LIN {X 0,Y 476.575,Z 542.325,A -85,B 0,C 180,E1 -7304.355,E2 -7304.355} C_VEL
LIN {X 0,Y 476.998,Z 529.723,A -85,B 0,C 180,E1 -7304.805,E2 -7304.805} C_VEL
LIN {X 0,Y 477.328,Z 516.997,A -85,B 0,C 180,E1 -7305.095,E2 -7305.095} C_VEL
LIN {X 0,Y 477.658,Z 432.911,A -85,B 0,C 180,E1 -7306.37,E2 -7306.37} C_VEL
LIN {X 0,Y 475.32,Z 411.409,A -85,B 0,C 180,E1 -7306.785,E2 -7306.785} C_VEL
LIN {X 0,Y 475.32,Z 409.484,A -85,B 0,C 180,E1 -7306.979,E2 -7306.979} C_VEL
LIN {X 0,Y 476.001,Z 385.629,A -85,B 0,C 180,E1 -7310.076,E2 -7310.076} C_VEL
LIN {X 0,Y 476.795,Z 363.158,A -85,B 0,C 180,E1 -7312.992,E2 -7312.992} C_VEL
LIN {X 0,Y 477.623,Z 341.029,A -85,B 0,C 180,E1 -7315.89,E2 -7315.89} C_VEL
LIN {X 0,Y 478.026,Z 328.359,A -85,B 0,C 180,E1 -7317.578,E2 -7317.578} C_VEL
LIN {X 0,Y 474.979,Z 313.924,A -85,B 0,C 180,E1 -7319.714,E2 -7319.714} C_VEL
LIN {X 0,Y 474.64,Z 312.462,A -85,B 0,C 180,E1 -7319.982,E2 -7319.982} C_VEL
LIN {X 0,Y 474.612,Z 312.36,A -85,B 0,C 180,E1 -7323.222,E2 -7323.222} C_VEL
LIN {X 0,Y 474.569,Z 312.369,A -85,B 0,C 180,E1 -7326.325,E2 -7326.325} C_VEL
LIN {X 0,Y 474.597,Z 312.358,A -85,B 0,C 180,E1 -7329.643,E2 -7329.643} C_VEL
LIN {X 0,Y 474.565,Z 312.367,A -85,B 0,C 180,E1 -7332.939,E2 -7332.939} C_VEL
LIN {X 0,Y 474.598,Z 312.354,A -85,B 0,C 180,E1 -7335.894,E2 -7335.894} C_VEL
LIN {X 0,Y 474.596,Z 312.364,A -85,B 0,C 180,E1 -7339.044,E2 -7339.044} C_VEL
LIN {X 0,Y 474.584,Z 312.349,A -85,B 0,C 180,E1 -7341.707,E2 -7341.707} C_VEL
LIN {X 0,Y 474.606,Z 312.35,A -85,B 0,C 180,E1 -7344.724,E2 -7344.724} C_VEL
LIN {X 0,Y 474.621,Z 312.366,A -85,B 0,C 180,E1 -7347.787,E2 -7347.787} C_VEL
LIN {X 0,Y 474.6,Z 312.355,A -85,B 0,C 180,E1 -7350.888,E2 -7350.888} C_VEL
LIN {X 0,Y 474.584,Z 312.366,A -85,B 0,C 180,E1 -7353.624,E2 -7353.624} C_VEL
LIN {X 0,Y 474.627,Z 312.357,A -85,B 0,C 180,E1 -7356.642,E2 -7356.642} C_VEL
LIN {X 0,Y 474.645,Z 312.353,A -85,B 0,C 180,E1 -7360.089,E2 -7360.089} C_VEL
LIN {X 0,Y 474.626,Z 312.359,A -85,B 0,C 180,E1 -7362.774,E2 -7362.774} C_VEL
LIN {X 0,Y 474.637,Z 312.361,A -85,B 0,C 180,E1 -7365.421,E2 -7365.421} C_VEL
LIN {X 0,Y 474.696,Z 312.353,A -85,B 0,C 180,E1 -7368.037,E2 -7368.037} C_VEL
LIN {X 0,Y 474.693,Z 312.356,A -85,B 0,C 180,E1 -7371.486,E2 -7371.486} C_VEL
LIN {X 0,Y 474.749,Z 312.343,A -85,B 0,C 180,E1 -7374.052,E2 -7374.052} C_VEL
LIN {X 0,Y 474.863,Z 312.335,A -85,B 0,C 180,E1 -7377.455,E2 -7377.455} C_VEL
LIN {X 0,Y 474.869,Z 312.325,A -85,B 0,C 180,E1 -7380,E2 -7380} C_VEL
LIN {X 0,Y 474.872,Z 312.326,A -85,B 0,C 180,E1 -7382.545,E2 -7382.545} C_VEL
LIN {X 0,Y 474.73,Z 312.346,A -85,B 0,C 180,E1 -7385.948,E2 -7385.948} C_VEL
LIN {X 0,Y 474.699,Z 312.345,A -85,B 0,C 180,E1 -7388.514,E2 -7388.514} C_VEL
LIN {X 0,Y 474.696,Z 312.352,A -85,B 0,C 180,E1 -7391.963,E2 -7391.963} C_VEL
LIN {X 0,Y 474.671,Z 312.357,A -85,B 0,C 180,E1 -7395.767,E2 -7395.767} C_VEL
LIN {X 0,Y 474.652,Z 312.357,A -85,B 0,C 180,E1 -7399.011,E2 -7399.011} C_VEL
LIN {X 0,Y 474.58,Z 312.368,A -85,B 0,C 180,E1 -7401.729,E2 -7401.729} C_VEL
LIN {X 0,Y 474.619,Z 312.36,A -85,B 0,C 180,E1 -7404.495,E2 -7404.495} C_VEL
LIN {X 0,Y 474.592,Z 312.36,A -85,B 0,C 180,E1 -7407.327,E2 -7407.327} C_VEL
LIN {X 0,Y 474.582,Z 312.348,A -85,B 0,C 180,E1 -7410.232,E2 -7410.232} C_VEL
LIN {X 0,Y 474.609,Z 312.362,A -85,B 0,C 180,E1 -7413.223,E2 -7413.223} C_VEL
LIN {X 0,Y 474.577,Z 312.363,A -85,B 0,C 180,E1 -7416.325,E2 -7416.325} C_VEL
LIN {X 0,Y 474.596,Z 312.354,A -85,B 0,C 180,E1 -7419.644,E2 -7419.644} C_VEL
LIN {X 0,Y 474.564,Z 312.369,A -85,B 0,C 180,E1 -7422.94,E2 -7422.94} C_VEL
LIN {X 0,Y 474.576,Z 312.358,A -85,B 0,C 180,E1 -7425.892,E2 -7425.892} C_VEL
LIN {X 0,Y 474.596,Z 312.364,A -85,B 0,C 180,E1 -7429.046,E2 -7429.046} C_VEL
LIN {X 0,Y 474.594,Z 312.36,A -85,B 0,C 180,E1 -7431.707,E2 -7431.707} C_VEL
LIN {X 0,Y 474.616,Z 312.362,A -85,B 0,C 180,E1 -7434.726,E2 -7434.726} C_VEL
LIN {X 0,Y 474.615,Z 312.362,A -85,B 0,C 180,E1 -7437.787,E2 -7437.787} C_VEL
LIN {X 0,Y 474.592,Z 312.366,A -85,B 0,C 180,E1 -7440.892,E2 -7440.892} C_VEL
LIN {X 0,Y 474.571,Z 312.359,A -85,B 0,C 180,E1 -7443.624,E2 -7443.624} C_VEL
LIN {X 0,Y 474.634,Z 312.361,A -85,B 0,C 180,E1 -7446.643,E2 -7446.643} C_VEL
LIN {X 0,Y 474.647,Z 312.359,A -85,B 0,C 180,E1 -7450.09,E2 -7450.09} C_VEL
LIN {X 0,Y 474.625,Z 312.333,A -85,B 0,C 180,E1 -7451.631,E2 -7451.631} C_VEL
LIN {X 0,Y 474.463,Z 312.988,A -85,B 0,C 180,E1 -7452.075,E2 -7452.075} C_VEL
LIN {X 0,Y 474.092,Z 314.652,A -85,B 0,C 180,E1 -7452.481,E2 -7452.481} C_VEL
LIN {X 0,Y 473.329,Z 318.415,A -85,B 0,C 180,E1 -7453.005,E2 -7453.005} C_VEL
LIN {X 0,Y 472.491,Z 323.287,A -85,B 0,C 180,E1 -7453.422,E2 -7453.422} C_VEL
LIN {X 0,Y 471.778,Z 328.831,A -85,B 0,C 180,E1 -7453.729,E2 -7453.729} C_VEL
LIN {X 0,Y 471.44,Z 334.777,A -85,B 0,C 180,E1 -7453.9,E2 -7453.9} C_VEL
LIN {X 0,Y 471.117,Z 394.353,A -85,B 0,C 180,E1 -7454.84,E2 -7454.84} C_VEL
LIN {X 0,Y 470.981,Z 407.411,A -85,B 0,C 180,E1 -7455.222,E2 -7455.222} C_VEL
LIN {X 0,Y 470.798,Z 419.402,A -85,B 0,C 180,E1 -7455.741,E2 -7455.741} C_VEL
LIN {X 0,Y 470.507,Z 431.055,A -85,B 0,C 180,E1 -7456.419,E2 -7456.419} C_VEL
LIN {X 0,Y 470.005,Z 442.247,A -85,B 0,C 180,E1 -7457.258,E2 -7457.258} C_VEL
LIN {X 0,Y 469.55,Z 452.592,A -85,B 0,C 180,E1 -7458.233,E2 -7458.233} C_VEL
LIN {X 0,Y 469.181,Z 461.025,A -85,B 0,C 180,E1 -7459.208,E2 -7459.208} C_VEL
LIN {X 0,Y 468.744,Z 468.789,A -85,B 0,C 180,E1 -7460.289,E2 -7460.289} C_VEL
LIN {X 0,Y 468.373,Z 476.47,A -85,B 0,C 180,E1 -7461.609,E2 -7461.609} C_VEL
LIN {X 0,Y 468.091,Z 482.229,A -85,B 0,C 180,E1 -7462.84,E2 -7462.84} C_VEL
LIN {X 0,Y 467.937,Z 486.507,A -85,B 0,C 180,E1 -7463.965,E2 -7463.965} C_VEL
LIN {X 0,Y 467.639,Z 490.4,A -85,B 0,C 180,E1 -7465.259,E2 -7465.259} C_VEL
LIN {X 0,Y 467.443,Z 493.271,A -85,B 0,C 180,E1 -7466.552,E2 -7466.552} C_VEL
LIN {X 0,Y 467.481,Z 494.631,A -85,B 0,C 180,E1 -7467.415,E2 -7467.415} C_VEL
LIN {X 0,Y 467.356,Z 495.617,A -85,B 0,C 180,E1 -7468.277,E2 -7468.277} C_VEL
LIN {X 0,Y 467.433,Z 496.204,A -85,B 0,C 180,E1 -7469.139,E2 -7469.139} C_VEL
LIN {X 0,Y 467.417,Z 496.436,A -85,B 0,C 180,E1 -7470,E2 -7470} C_VEL
LIN {X 0,Y 467.433,Z 496.253,A -85,B 0,C 180,E1 -7470.861,E2 -7470.861} C_VEL
LIN {X 0,Y 467.356,Z 495.698,A -85,B 0,C 180,E1 -7471.723,E2 -7471.723} C_VEL
LIN {X 0,Y 467.48,Z 494.743,A -85,B 0,C 180,E1 -7472.585,E2 -7472.585} C_VEL
LIN {X 0,Y 467.437,Z 493.435,A -85,B 0,C 180,E1 -7473.448,E2 -7473.448} C_VEL
LIN {X 0,Y 467.634,Z 490.625,A -85,B 0,C 180,E1 -7474.741,E2 -7474.741} C_VEL
LIN {X 0,Y 467.927,Z 486.808,A -85,B 0,C 180,E1 -7476.035,E2 -7476.035} C_VEL
LIN {X 0,Y 468.063,Z 481.73,A -85,B 0,C 180,E1 -7477.377,E2 -7477.377} C_VEL
LIN {X 0,Y 468.507,Z 474.508,A -85,B 0,C 180,E1 -7478.845,E2 -7478.845} C_VEL
LIN {X 0,Y 468.968,Z 466.485,A -85,B 0,C 180,E1 -7480.142,E2 -7480.142} C_VEL
LIN {X 0,Y 469.344,Z 458.267,A -85,B 0,C 180,E1 -7481.225,E2 -7481.225} C_VEL
LIN {X 0,Y 469.747,Z 449.245,A -85,B 0,C 180,E1 -7482.2,E2 -7482.2} C_VEL
LIN {X 0,Y 470.256,Z 438.755,A -85,B 0,C 180,E1 -7483.114,E2 -7483.114} C_VEL
LIN {X 0,Y 470.569,Z 427.264,A -85,B 0,C 180,E1 -7483.914,E2 -7483.914} C_VEL
LIN {X 0,Y 470.826,Z 416.033,A -85,B 0,C 180,E1 -7484.517,E2 -7484.517} C_VEL
LIN {X 0,Y 471.032,Z 402.87,A -85,B 0,C 180,E1 -7485.025,E2 -7485.025} C_VEL
LIN {X 0,Y 471.056,Z 389.173,A -85,B 0,C 180,E1 -7485.356,E2 -7485.356} C_VEL
LIN {X 0,Y 471.439,Z 324.141,A -85,B 0,C 180,E1 -7486.359,E2 -7486.359} C_VEL
LIN {X 0,Y 467.78,Z 314.282,A -85,B 0,C 180,E1 -7486.672,E2 -7486.672} C_VEL
LIN {X 0,Y 467.575,Z 313.366,A -85,B 0,C 180,E1 -7486.826,E2 -7486.826} C_VEL
LIN {X 0,Y 467.589,Z 313.223,A -85,B 0,C 180,E1 -7489.309,E2 -7489.309} C_VEL
LIN {X 0,Y 467.529,Z 313.235,A -85,B 0,C 180,E1 -7492.074,E2 -7492.074} C_VEL
LIN {X 0,Y 467.549,Z 313.246,A -85,B 0,C 180,E1 -7494.89,E2 -7494.89} C_VEL
LIN {X 0,Y 467.54,Z 313.225,A -85,B 0,C 180,E1 -7497.774,E2 -7497.774} C_VEL
LIN {X 0,Y 467.534,Z 313.246,A -85,B 0,C 180,E1 -7501.037,E2 -7501.037} C_VEL
LIN {X 0,Y 467.563,Z 313.241,A -85,B 0,C 180,E1 -7504.237,E2 -7504.237} C_VEL
LIN {X 0,Y 467.519,Z 313.239,A -85,B 0,C 180,E1 -7507.181,E2 -7507.181} C_VEL
LIN {X 0,Y 467.553,Z 313.244,A -85,B 0,C 180,E1 -7510.266,E2 -7510.266} C_VEL
LIN {X 0,Y 467.513,Z 313.241,A -85,B 0,C 180,E1 -7512.568,E2 -7512.568} C_VEL
LIN {X 0,Y 467.558,Z 313.243,A -85,B 0,C 180,E1 -7515.051,E2 -7515.051} C_VEL
LIN {X 0,Y 467.555,Z 313.239,A -85,B 0,C 180,E1 -7518.725,E2 -7518.725} C_VEL
LIN {X 0,Y 467.546,Z 313.229,A -85,B 0,C 180,E1 -7521.953,E2 -7521.953} C_VEL
LIN {X 0,Y 467.548,Z 313.243,A -85,B 0,C 180,E1 -7525.166,E2 -7525.166} C_VEL
LIN {X 0,Y 467.568,Z 313.236,A -85,B 0,C 180,E1 -7528.259,E2 -7528.259} C_VEL
LIN {X 0,Y 467.533,Z 313.226,A -85,B 0,C 180,E1 -7531.247,E2 -7531.247} C_VEL
LIN {X 0,Y 467.571,Z 313.24,A -85,B 0,C 180,E1 -7534.4,E2 -7534.4} C_VEL
LIN {X 0,Y 467.543,Z 313.242,A -85,B 0,C 180,E1 -7536.994,E2 -7536.994} C_VEL
LIN {X 0,Y 467.6,Z 313.229,A -85,B 0,C 180,E1 -7539.776,E2 -7539.776} C_VEL
LIN {X 0,Y 467.574,Z 313.245,A -85,B 0,C 180,E1 -7542.505,E2 -7542.505} C_VEL
LIN {X 0,Y 467.585,Z 313.228,A -85,B 0,C 180,E1 -7545.196,E2 -7545.196} C_VEL
LIN {X 0,Y 467.648,Z 313.229,A -85,B 0,C 180,E1 -7547.854,E2 -7547.854} C_VEL
LIN {X 0,Y 467.626,Z 313.225,A -85,B 0,C 180,E1 -7551.356,E2 -7551.356} C_VEL
LIN {X 0,Y 467.684,Z 313.223,A -85,B 0,C 180,E1 -7553.962,E2 -7553.962} C_VEL
LIN {X 0,Y 467.813,Z 313.206,A -85,B 0,C 180,E1 -7557.417,E2 -7557.417} C_VEL
LIN {X 0,Y 467.838,Z 313.2,A -85,B 0,C 180,E1 -7560,E2 -7560} C_VEL
LIN {X 0,Y 467.803,Z 313.213,A -85,B 0,C 180,E1 -7562.583,E2 -7562.583} C_VEL
LIN {X 0,Y 467.713,Z 313.218,A -85,B 0,C 180,E1 -7566.038,E2 -7566.038} C_VEL
LIN {X 0,Y 467.65,Z 313.232,A -85,B 0,C 180,E1 -7568.643,E2 -7568.643} C_VEL
LIN {X 0,Y 467.64,Z 313.228,A -85,B 0,C 180,E1 -7572.354,E2 -7572.354} C_VEL
LIN {X 0,Y 467.641,Z 313.232,A -85,B 0,C 180,E1 -7575.885,E2 -7575.885} C_VEL
LIN {X 0,Y 467.612,Z 313.225,A -85,B 0,C 180,E1 -7579.308,E2 -7579.308} C_VEL
LIN {X 0,Y 467.527,Z 313.238,A -85,B 0,C 180,E1 -7582.074,E2 -7582.074} C_VEL
LIN {X 0,Y 467.552,Z 313.241,A -85,B 0,C 180,E1 -7584.89,E2 -7584.89} C_VEL
LIN {X 0,Y 467.571,Z 313.236,A -85,B 0,C 180,E1 -7587.772,E2 -7587.772} C_VEL
LIN {X 0,Y 467.561,Z 313.24,A -85,B 0,C 180,E1 -7591.045,E2 -7591.045} C_VEL
LIN {X 0,Y 467.569,Z 313.237,A -85,B 0,C 180,E1 -7594.24,E2 -7594.24} C_VEL
LIN {X 0,Y 467.51,Z 313.246,A -85,B 0,C 180,E1 -7597.181,E2 -7597.181} C_VEL
LIN {X 0,Y 467.552,Z 313.245,A -85,B 0,C 180,E1 -7600.267,E2 -7600.267} C_VEL
LIN {X 0,Y 467.542,Z 313.238,A -85,B 0,C 180,E1 -7603.746,E2 -7603.746} C_VEL
LIN {X 0,Y 467.529,Z 313.239,A -85,B 0,C 180,E1 -7606.253,E2 -7606.253} C_VEL
LIN {X 0,Y 467.553,Z 313.238,A -85,B 0,C 180,E1 -7609.734,E2 -7609.734} C_VEL
LIN {X 0,Y 467.513,Z 313.248,A -85,B 0,C 180,E1 -7612.82,E2 -7612.82} C_VEL
LIN {X 0,Y 467.573,Z 313.244,A -85,B 0,C 180,E1 -7615.761,E2 -7615.761} C_VEL
LIN {X 0,Y 467.542,Z 313.24,A -85,B 0,C 180,E1 -7618.961,E2 -7618.961} C_VEL
LIN {X 0,Y 467.61,Z 313.465,A -85,B 0,C 180,E1 -7619.816,E2 -7619.816} C_VEL
LIN {X 0,Y 470.901,Z 328.362,A -85,B 0,C 180,E1 -7622.091,E2 -7622.091} C_VEL
LIN {X 0,Y 471.126,Z 332.687,A -85,B 0,C 180,E1 -7622.697,E2 -7622.697} C_VEL
LIN {X 0,Y 470.179,Z 355.502,A -85,B 0,C 180,E1 -7625.755,E2 -7625.755} C_VEL
LIN {X 0,Y 469.304,Z 378.017,A -85,B 0,C 180,E1 -7628.731,E2 -7628.731} C_VEL
LIN {X 0,Y 468.526,Z 401.754,A -85,B 0,C 180,E1 -7631.865,E2 -7631.865} C_VEL
LIN {X 0,Y 468.274,Z 409.892,A -85,B 0,C 180,E1 -7632.926,E2 -7632.926} C_VEL
LIN {X 0,Y 470.965,Z 436.984,A -85,B 0,C 180,E1 -7633.468,E2 -7633.468} C_VEL
LIN {X 0,Y 470.367,Z 520.419,A -85,B 0,C 180,E1 -7634.759,E2 -7634.759} C_VEL
LIN {X 0,Y 469.932,Z 533.749,A -85,B 0,C 180,E1 -7635.133,E2 -7635.133} C_VEL
LIN {X 0,Y 469.454,Z 545.997,A -85,B 0,C 180,E1 -7635.644,E2 -7635.644} C_VEL
LIN {X 0,Y 468.869,Z 558.388,A -85,B 0,C 180,E1 -7636.345,E2 -7636.345} C_VEL
LIN {X 0,Y 468.42,Z 569.231,A -85,B 0,C 180,E1 -7637.139,E2 -7637.139} C_VEL
LIN {X 0,Y 468.006,Z 579.654,A -85,B 0,C 180,E1 -7638.084,E2 -7638.084} C_VEL
LIN {X 0,Y 467.552,Z 589.428,A -85,B 0,C 180,E1 -7639.17,E2 -7639.17} C_VEL
LIN {X 0,Y 467.242,Z 597.469,A -85,B 0,C 180,E1 -7640.258,E2 -7640.258} C_VEL
LIN {X 0,Y 467.094,Z 605.36,A -85,B 0,C 180,E1 -7641.564,E2 -7641.564} C_VEL
LIN {X 0,Y 466.941,Z 612.637,A -85,B 0,C 180,E1 -7643.084,E2 -7643.084} C_VEL
LIN {X 0,Y 466.958,Z 617.503,A -85,B 0,C 180,E1 -7644.386,E2 -7644.386} C_VEL
LIN {X 0,Y 467.026,Z 621.231,A -85,B 0,C 180,E1 -7645.685,E2 -7645.685} C_VEL
LIN {X 0,Y 467.023,Z 623.15,A -85,B 0,C 180,E1 -7646.549,E2 -7646.549} C_VEL
LIN {X 0,Y 467.006,Z 624.588,A -85,B 0,C 180,E1 -7647.412,E2 -7647.412} C_VEL
LIN {X 0,Y 467.132,Z 626.26,A -85,B 0,C 180,E1 -7649.138,E2 -7649.138} C_VEL
LIN {X 0,Y 467.123,Z 626.482,A -85,B 0,C 180,E1 -7650,E2 -7650} C_VEL
LIN {X 0,Y 467.132,Z 626.26,A -85,B 0,C 180,E1 -7650.862,E2 -7650.862} C_VEL
LIN {X 0,Y 467.006,Z 624.591,A -85,B 0,C 180,E1 -7652.588,E2 -7652.588} C_VEL
LIN {X 0,Y 467.023,Z 623.154,A -85,B 0,C 180,E1 -7653.451,E2 -7653.451} C_VEL
LIN {X 0,Y 466.997,Z 620.126,A -85,B 0,C 180,E1 -7654.748,E2 -7654.748} C_VEL
LIN {X 0,Y 467.001,Z 614.792,A -85,B 0,C 180,E1 -7656.377,E2 -7656.377} C_VEL
LIN {X 0,Y 467.01,Z 608.704,A -85,B 0,C 180,E1 -7657.784,E2 -7657.784} C_VEL
LIN {X 0,Y 467.155,Z 601.63,A -85,B 0,C 180,E1 -7659.089,E2 -7659.089} C_VEL
LIN {X 0,Y 467.419,Z 592.804,A -85,B 0,C 180,E1 -7660.395,E2 -7660.395} C_VEL
LIN {X 0,Y 467.744,Z 583.782,A -85,B 0,C 180,E1 -7661.483,E2 -7661.483} C_VEL
LIN {X 0,Y 468.234,Z 574.725,A -85,B 0,C 180,E1 -7662.386,E2 -7662.386} C_VEL
LIN {X 0,Y 468.652,Z 563.142,A -85,B 0,C 180,E1 -7663.33,E2 -7663.33} C_VEL
LIN {X 0,Y 469.224,Z 551.148,A -85,B 0,C 180,E1 -7664.086,E2 -7664.086} C_VEL
LIN {X 0,Y 469.764,Z 538.709,A -85,B 0,C 180,E1 -7664.678,E2 -7664.678} C_VEL
LIN {X 0,Y 470.233,Z 525.972,A -85,B 0,C 180,E1 -7665.106,E2 -7665.106} C_VEL
LIN {X 0,Y 470.503,Z 512.684,A -85,B 0,C 180,E1 -7665.375,E2 -7665.375} C_VEL
LIN {X 0,Y 470.882,Z 434.034,A -85,B 0,C 180,E1 -7666.579,E2 -7666.579} C_VEL
LIN {X 0,Y 468.293,Z 410.384,A -85,B 0,C 180,E1 -7667.045,E2 -7667.045} C_VEL
LIN {X 0,Y 468.312,Z 408.488,A -85,B 0,C 180,E1 -7667.241,E2 -7667.241} C_VEL
LIN {X 0,Y 469.056,Z 384.679,A -85,B 0,C 180,E1 -7670.387,E2 -7670.387} C_VEL
LIN {X 0,Y 469.821,Z 363.974,A -85,B 0,C 180,E1 -7673.12,E2 -7673.12} C_VEL
LIN {X 0,Y 470.704,Z 341.88,A -85,B 0,C 180,E1 -7676.061,E2 -7676.061} C_VEL
LIN {X 0,Y 471.108,Z 329.625,A -85,B 0,C 180,E1 -7677.721,E2 -7677.721} C_VEL
LIN {X 0,Y 467.711,Z 313.916,A -85,B 0,C 180,E1 -7680.099,E2 -7680.099} C_VEL
LIN {X 0,Y 467.596,Z 313.339,A -85,B 0,C 180,E1 -7680.232,E2 -7680.232} C_VEL
LIN {X 0,Y 467.571,Z 313.236,A -85,B 0,C 180,E1 -7682.759,E2 -7682.759} C_VEL
LIN {X 0,Y 467.541,Z 313.24,A -85,B 0,C 180,E1 -7685.89,E2 -7685.89} C_VEL
LIN {X 0,Y 467.54,Z 313.238,A -85,B 0,C 180,E1 -7689.148,E2 -7689.148} C_VEL
LIN {X 0,Y 467.555,Z 313.242,A -85,B 0,C 180,E1 -7691.404,E2 -7691.404} C_VEL
LIN {X 0,Y 467.561,Z 313.222,A -85,B 0,C 180,E1 -7695.052,E2 -7695.052} C_VEL
LIN {X 0,Y 467.557,Z 313.241,A -85,B 0,C 180,E1 -7698.725,E2 -7698.725} C_VEL
LIN {X 0,Y 467.535,Z 313.221,A -85,B 0,C 180,E1 -7701.952,E2 -7701.952} C_VEL
LIN {X 0,Y 467.545,Z 313.23,A -85,B 0,C 180,E1 -7705.166,E2 -7705.166} C_VEL
LIN {X 0,Y 467.572,Z 313.241,A -85,B 0,C 180,E1 -7708.259,E2 -7708.259} C_VEL
LIN {X 0,Y 467.547,Z 313.235,A -85,B 0,C 180,E1 -7711.248,E2 -7711.248} C_VEL
LIN {X 0,Y 467.56,Z 313.244,A -85,B 0,C 180,E1 -7714.157,E2 -7714.157} C_VEL
LIN {X 0,Y 467.569,Z 313.236,A -85,B 0,C 180,E1 -7716.995,E2 -7716.995} C_VEL
LIN {X 0,Y 467.614,Z 313.224,A -85,B 0,C 180,E1 -7719.777,E2 -7719.777} C_VEL
LIN {X 0,Y 467.586,Z 313.236,A -85,B 0,C 180,E1 -7722.506,E2 -7722.506} C_VEL
LIN {X 0,Y 467.596,Z 313.236,A -85,B 0,C 180,E1 -7725.196,E2 -7725.196} C_VEL
LIN {X 0,Y 467.648,Z 313.229,A -85,B 0,C 180,E1 -7727.854,E2 -7727.854} C_VEL
LIN {X 0,Y 467.652,Z 313.231,A -85,B 0,C 180,E1 -7731.357,E2 -7731.357} C_VEL
LIN {X 0,Y 467.714,Z 313.219,A -85,B 0,C 180,E1 -7733.962,E2 -7733.962} C_VEL
LIN {X 0,Y 467.804,Z 313.213,A -85,B 0,C 180,E1 -7737.417,E2 -7737.417} C_VEL
LIN {X 0,Y 467.839,Z 313.2,A -85,B 0,C 180,E1 -7740,E2 -7740} C_VEL
LIN {X 0,Y 467.814,Z 313.206,A -85,B 0,C 180,E1 -7742.583,E2 -7742.583} C_VEL
LIN {X 0,Y 467.695,Z 313.222,A -85,B 0,C 180,E1 -7746.038,E2 -7746.038} C_VEL
LIN {X 0,Y 467.658,Z 313.221,A -85,B 0,C 180,E1 -7748.643,E2 -7748.643} C_VEL
LIN {X 0,Y 467.648,Z 313.228,A -85,B 0,C 180,E1 -7752.146,E2 -7752.146} C_VEL
LIN {X 0,Y 467.629,Z 313.233,A -85,B 0,C 180,E1 -7755.695,E2 -7755.695} C_VEL
LIN {X 0,Y 467.611,Z 313.237,A -85,B 0,C 180,E1 -7759.308,E2 -7759.308} C_VEL
LIN {X 0,Y 467.523,Z 313.244,A -85,B 0,C 180,E1 -7762.075,E2 -7762.075} C_VEL
LIN {X 0,Y 467.552,Z 313.242,A -85,B 0,C 180,E1 -7764.89,E2 -7764.89} C_VEL
LIN {X 0,Y 467.538,Z 313.23,A -85,B 0,C 180,E1 -7767.774,E2 -7767.774} C_VEL
LIN {X 0,Y 467.539,Z 313.227,A -85,B 0,C 180,E1 -7771.041,E2 -7771.041} C_VEL
LIN {X 0,Y 467.57,Z 313.239,A -85,B 0,C 180,E1 -7774.24,E2 -7774.24} C_VEL
LIN {X 0,Y 467.533,Z 313.244,A -85,B 0,C 180,E1 -7777.185,E2 -7777.185} C_VEL
LIN {X 0,Y 467.551,Z 313.232,A -85,B 0,C 180,E1 -7780.268,E2 -7780.268} C_VEL
LIN {X 0,Y 467.54,Z 313.245,A -85,B 0,C 180,E1 -7783.747,E2 -7783.747} C_VEL
LIN {X 0,Y 467.525,Z 313.233,A -85,B 0,C 180,E1 -7786.253,E2 -7786.253} C_VEL
LIN {X 0,Y 467.557,Z 313.238,A -85,B 0,C 180,E1 -7788.727,E2 -7788.727} C_VEL
LIN {X 0,Y 467.544,Z 313.236,A -85,B 0,C 180,E1 -7791.954,E2 -7791.954} C_VEL
LIN {X 0,Y 467.554,Z 313.246,A -85,B 0,C 180,E1 -7795.167,E2 -7795.167} C_VEL
LIN {X 0,Y 467.547,Z 313.24,A -85,B 0,C 180,E1 -7798.258,E2 -7798.258} C_VEL
LIN {X 0,Y 467.538,Z 313.236,A -85,B 0,C 180,E1 -7801.248,E2 -7801.248} C_VEL
LIN {X 0,Y 467.561,Z 313.24,A -85,B 0,C 180,E1 -7804.406,E2 -7804.406} C_VEL
LIN {X 0,Y 467.572,Z 313.235,A -85,B 0,C 180,E1 -7806.996,E2 -7806.996} C_VEL
LIN {X 0,Y 467.618,Z 313.237,A -85,B 0,C 180,E1 -7809.777,E2 -7809.777} C_VEL
LIN {X 0,Y 467.564,Z 313.194,A -85,B 0,C 180,E1 -7812.956,E2 -7812.956} C_VEL
LIN {X 0,Y 467.652,Z 313.605,A -85,B 0,C 180,E1 -7813.339,E2 -7813.339} C_VEL
LIN {X 0,Y 468.05,Z 315.073,A -85,B 0,C 180,E1 -7813.458,E2 -7813.458} C_VEL
LIN {X 0,Y 471.58,Z 324.691,A -85,B 0,C 180,E1 -7813.748,E2 -7813.748} C_VEL
LIN {X 0,Y 471.44,Z 334.777,A -85,B 0,C 180,E1 -7813.9,E2 -7813.9} C_VEL
LIN {X 0,Y 470.741,Z 340.627,A -85,B 0,C 180,E1 -7813.965,E2 -7813.965} C_VEL
LIN {X 0,Y 465.07,Z 359.64,A -85,B 0,C 180,E1 -7814.052,E2 -7814.052} C_VEL
LIN {X 0,Y 464.435,Z 365.486,A -85,B 0,C 180,E1 -7814.12,E2 -7814.12} C_VEL
LIN {X 0,Y 464.316,Z 395.352,A -85,B 0,C 180,E1 -7814.612,E2 -7814.612} C_VEL
LIN {X 0,Y 464.175,Z 408.403,A -85,B 0,C 180,E1 -7815.001,E2 -7815.001} C_VEL
LIN {X 0,Y 463.987,Z 420.389,A -85,B 0,C 180,E1 -7815.528,E2 -7815.528} C_VEL
LIN {X 0,Y 463.685,Z 431.642,A -85,B 0,C 180,E1 -7816.188,E2 -7816.188} C_VEL
LIN {X 0,Y 463.15,Z 443.231,A -85,B 0,C 180,E1 -7817.067,E2 -7817.067} C_VEL
LIN {X 0,Y 462.67,Z 453.574,A -85,B 0,C 180,E1 -7818.056,E2 -7818.056} C_VEL
LIN {X 0,Y 462.278,Z 462.006,A -85,B 0,C 180,E1 -7819.045,E2 -7819.045} C_VEL
LIN {X 0,Y 461.821,Z 469.769,A -85,B 0,C 180,E1 -7820.142,E2 -7820.142} C_VEL
LIN {X 0,Y 461.422,Z 477.451,A -85,B 0,C 180,E1 -7821.482,E2 -7821.482} C_VEL
LIN {X 0,Y 461.119,Z 483.209,A -85,B 0,C 180,E1 -7822.731,E2 -7822.731} C_VEL
LIN {X 0,Y 460.953,Z 487.486,A -85,B 0,C 180,E1 -7823.873,E2 -7823.873} C_VEL
LIN {X 0,Y 460.632,Z 491.379,A -85,B 0,C 180,E1 -7825.186,E2 -7825.186} C_VEL
LIN {X 0,Y 460.423,Z 494.25,A -85,B 0,C 180,E1 -7826.5,E2 -7826.5} C_VEL
LIN {X 0,Y 460.464,Z 495.609,A -85,B 0,C 180,E1 -7827.376,E2 -7827.376} C_VEL
LIN {X 0,Y 460.335,Z 496.595,A -85,B 0,C 180,E1 -7828.25,E2 -7828.25} C_VEL
LIN {X 0,Y 460.413,Z 497.181,A -85,B 0,C 180,E1 -7829.125,E2 -7829.125} C_VEL
LIN {X 0,Y 460.397,Z 497.413,A -85,B 0,C 180,E1 -7830,E2 -7830} C_VEL
LIN {X 0,Y 460.412,Z 497.23,A -85,B 0,C 180,E1 -7830.875,E2 -7830.875} C_VEL
LIN {X 0,Y 460.335,Z 496.675,A -85,B 0,C 180,E1 -7831.75,E2 -7831.75} C_VEL
LIN {X 0,Y 460.463,Z 495.72,A -85,B 0,C 180,E1 -7832.624,E2 -7832.624} C_VEL
LIN {X 0,Y 460.418,Z 494.412,A -85,B 0,C 180,E1 -7833.5,E2 -7833.5} C_VEL
LIN {X 0,Y 460.627,Z 491.602,A -85,B 0,C 180,E1 -7834.814,E2 -7834.814} C_VEL
LIN {X 0,Y 460.941,Z 487.784,A -85,B 0,C 180,E1 -7836.127,E2 -7836.127} C_VEL
LIN {X 0,Y 461.094,Z 482.707,A -85,B 0,C 180,E1 -7837.488,E2 -7837.488} C_VEL
LIN {X 0,Y 461.568,Z 475.483,A -85,B 0,C 180,E1 -7838.979,E2 -7838.979} C_VEL
LIN {X 0,Y 462.055,Z 467.46,A -85,B 0,C 180,E1 -7840.295,E2 -7840.295} C_VEL
LIN {X 0,Y 462.45,Z 459.242,A -85,B 0,C 180,E1 -7841.394,E2 -7841.394} C_VEL
LIN {X 0,Y 462.882,Z 450.218,A -85,B 0,C 180,E1 -7842.384,E2 -7842.384} C_VEL
LIN {X 0,Y 463.414,Z 439.727,A -85,B 0,C 180,E1 -7843.311,E2 -7843.311} C_VEL
LIN {X 0,Y 463.75,Z 428.235,A -85,B 0,C 180,E1 -7844.123,E2 -7844.123} C_VEL
LIN {X 0,Y 464.019,Z 417.003,A -85,B 0,C 180,E1 -7844.735,E2 -7844.735} C_VEL
LIN {X 0,Y 464.23,Z 403.837,A -85,B 0,C 180,E1 -7845.25,E2 -7845.25} C_VEL
LIN {X 0,Y 464.249,Z 390.132,A -85,B 0,C 180,E1 -7845.587,E2 -7845.587} C_VEL
LIN {X 0,Y 464.739,Z 326.152,A -85,B 0,C 180,E1 -7846.585,E2 -7846.585} C_VEL
LIN {X 0,Y 460.728,Z 315.162,A -85,B 0,C 180,E1 -7846.937,E2 -7846.937} C_VEL
LIN {X 0,Y 460.544,Z 314.268,A -85,B 0,C 180,E1 -7847.083,E2 -7847.083} C_VEL
LIN {X 0,Y 460.544,Z 314.11,A -85,B 0,C 180,E1 -7849.616,E2 -7849.616} C_VEL
LIN {X 0,Y 460.506,Z 314.108,A -85,B 0,C 180,E1 -7852.428,E2 -7852.428} C_VEL
LIN {X 0,Y 460.509,Z 314.118,A -85,B 0,C 180,E1 -7855.297,E2 -7855.297} C_VEL
LIN {X 0,Y 460.502,Z 314.103,A -85,B 0,C 180,E1 -7858.236,E2 -7858.236} C_VEL
LIN {X 0,Y 460.494,Z 314.121,A -85,B 0,C 180,E1 -7861.277,E2 -7861.277} C_VEL
LIN {X 0,Y 460.511,Z 314.122,A -85,B 0,C 180,E1 -7864.501,E2 -7864.501} C_VEL
LIN {X 0,Y 460.484,Z 314.113,A -85,B 0,C 180,E1 -7867.624,E2 -7867.624} C_VEL
LIN {X 0,Y 460.511,Z 314.119,A -85,B 0,C 180,E1 -7871.013,E2 -7871.013} C_VEL
LIN {X 0,Y 460.506,Z 314.115,A -85,B 0,C 180,E1 -7874.589,E2 -7874.589} C_VEL
LIN {X 0,Y 460.469,Z 314.124,A -85,B 0,C 180,E1 -7877.812,E2 -7877.812} C_VEL
LIN {X 0,Y 460.505,Z 314.11,A -85,B 0,C 180,E1 -7880.135,E2 -7880.135} C_VEL
LIN {X 0,Y 460.464,Z 314.121,A -85,B 0,C 180,E1 -7883.469,E2 -7883.469} C_VEL
LIN {X 0,Y 460.511,Z 314.12,A -85,B 0,C 180,E1 -7886.673,E2 -7886.673} C_VEL
LIN {X 0,Y 460.49,Z 314.102,A -85,B 0,C 180,E1 -7889.758,E2 -7889.758} C_VEL
LIN {X 0,Y 460.484,Z 314.116,A -85,B 0,C 180,E1 -7892.75,E2 -7892.75} C_VEL
LIN {X 0,Y 460.508,Z 314.118,A -85,B 0,C 180,E1 -7895.666,E2 -7895.666} C_VEL
LIN {X 0,Y 460.51,Z 314.117,A -85,B 0,C 180,E1 -7898.58,E2 -7898.58} C_VEL
LIN {X 0,Y 460.574,Z 314.11,A -85,B 0,C 180,E1 -7901.31,E2 -7901.31} C_VEL
LIN {X 0,Y 460.578,Z 314.111,A -85,B 0,C 180,E1 -7904.058,E2 -7904.058} C_VEL
LIN {X 0,Y 460.601,Z 314.105,A -85,B 0,C 180,E1 -7907.666,E2 -7907.666} C_VEL
LIN {X 0,Y 460.582,Z 314.103,A -85,B 0,C 180,E1 -7911.223,E2 -7911.223} C_VEL
LIN {X 0,Y 460.651,Z 314.098,A -85,B 0,C 180,E1 -7913.869,E2 -7913.869} C_VEL
LIN {X 0,Y 460.758,Z 314.085,A -85,B 0,C 180,E1 -7917.377,E2 -7917.377} C_VEL
LIN {X 0,Y 460.787,Z 314.078,A -85,B 0,C 180,E1 -7920,E2 -7920} C_VEL
LIN {X 0,Y 460.747,Z 314.092,A -85,B 0,C 180,E1 -7922.623,E2 -7922.623} C_VEL
LIN {X 0,Y 460.679,Z 314.094,A -85,B 0,C 180,E1 -7926.13,E2 -7926.13} C_VEL
LIN {X 0,Y 460.598,Z 314.109,A -85,B 0,C 180,E1 -7928.777,E2 -7928.777} C_VEL
LIN {X 0,Y 460.589,Z 314.105,A -85,B 0,C 180,E1 -7932.435,E2 -7932.435} C_VEL
LIN {X 0,Y 460.594,Z 314.112,A -85,B 0,C 180,E1 -7935.998,E2 -7935.998} C_VEL
LIN {X 0,Y 460.559,Z 314.105,A -85,B 0,C 180,E1 -7939.616,E2 -7939.616} C_VEL
LIN {X 0,Y 460.503,Z 314.119,A -85,B 0,C 180,E1 -7942.429,E2 -7942.429} C_VEL
LIN {X 0,Y 460.528,Z 314.119,A -85,B 0,C 180,E1 -7945.794,E2 -7945.794} C_VEL
LIN {X 0,Y 460.518,Z 314.112,A -85,B 0,C 180,E1 -7948.235,E2 -7948.235} C_VEL
LIN {X 0,Y 460.514,Z 314.118,A -85,B 0,C 180,E1 -7951.283,E2 -7951.283} C_VEL
LIN {X 0,Y 460.513,Z 314.115,A -85,B 0,C 180,E1 -7954.503,E2 -7954.503} C_VEL
LIN {X 0,Y 460.477,Z 314.125,A -85,B 0,C 180,E1 -7957.626,E2 -7957.626} C_VEL
LIN {X 0,Y 460.511,Z 314.118,A -85,B 0,C 180,E1 -7961.014,E2 -7961.014} C_VEL
LIN {X 0,Y 460.506,Z 314.101,A -85,B 0,C 180,E1 -7964.59,E2 -7964.59} C_VEL
LIN {X 0,Y 460.47,Z 314.128,A -85,B 0,C 180,E1 -7967.814,E2 -7967.814} C_VEL
LIN {X 0,Y 460.506,Z 314.112,A -85,B 0,C 180,E1 -7970.136,E2 -7970.136} C_VEL
LIN {X 0,Y 460.456,Z 314.127,A -85,B 0,C 180,E1 -7973.469,E2 -7973.469} C_VEL
LIN {X 0,Y 460.514,Z 314.116,A -85,B 0,C 180,E1 -7976.675,E2 -7976.675} C_VEL
LIN {X 0,Y 460.562,Z 314.283,A -85,B 0,C 180,E1 -7979.543,E2 -7979.543} C_VEL
LIN {X 0,Y 463.698,Z 328.441,A -85,B 0,C 180,E1 -7981.759,E2 -7981.759} C_VEL
LIN {X 0,Y 464.298,Z 331.811,A -85,B 0,C 180,E1 -7982.261,E2 -7982.261} C_VEL
LIN {X 0,Y 463.38,Z 353.835,A -85,B 0,C 180,E1 -7985.271,E2 -7985.271} C_VEL
LIN {X 0,Y 462.374,Z 377.368,A -85,B 0,C 180,E1 -7988.436,E2 -7988.436} C_VEL
LIN {X 0,Y 461.491,Z 402.456,A -85,B 0,C 180,E1 -7991.809,E2 -7991.809} C_VEL
LIN {X 0,Y 461.293,Z 408.943,A -85,B 0,C 180,E1 -7992.663,E2 -7992.663} C_VEL
LIN {X 0,Y 464.154,Z 436.316,A -85,B 0,C 180,E1 -7993.223,E2 -7993.223} C_VEL
LIN {X 0,Y 463.521,Z 519.441,A -85,B 0,C 180,E1 -7994.529,E2 -7994.529} C_VEL
LIN {X 0,Y 463.065,Z 532.767,A -85,B 0,C 180,E1 -7994.907,E2 -7994.907} C_VEL
LIN {X 0,Y 462.499,Z 546.141,A -85,B 0,C 180,E1 -7995.48,E2 -7995.48} C_VEL
LIN {X 0,Y 461.903,Z 557.393,A -85,B 0,C 180,E1 -7996.135,E2 -7996.135} C_VEL
LIN {X 0,Y 461.393,Z 568.84,A -85,B 0,C 180,E1 -7996.991,E2 -7996.991} C_VEL
LIN {X 0,Y 460.954,Z 579.748,A -85,B 0,C 180,E1 -7998.011,E2 -7998.011} C_VEL
LIN {X 0,Y 460.514,Z 588.433,A -85,B 0,C 180,E1 -7999.003,E2 -7999.003} C_VEL
LIN {X 0,Y 460.174,Z 596.472,A -85,B 0,C 180,E1 -8000.107,E2 -8000.107} C_VEL
LIN {X 0,Y 460.007,Z 604.364,A -85,B 0,C 180,E1 -8001.433,E2 -8001.433} C_VEL
LIN {X 0,Y 459.885,Z 611.649,A -85,B 0,C 180,E1 -8002.978,E2 -8002.978} C_VEL
LIN {X 0,Y 459.902,Z 616.517,A -85,B 0,C 180,E1 -8004.3,E2 -8004.3} C_VEL
LIN {X 0,Y 459.967,Z 620.247,A -85,B 0,C 180,E1 -8005.619,E2 -8005.619} C_VEL
LIN {X 0,Y 459.976,Z 622.168,A -85,B 0,C 180,E1 -8006.496,E2 -8006.496} C_VEL
LIN {X 0,Y 459.961,Z 623.607,A -85,B 0,C 180,E1 -8007.373,E2 -8007.373} C_VEL
LIN {X 0,Y 460.108,Z 625.283,A -85,B 0,C 180,E1 -8009.125,E2 -8009.125} C_VEL
LIN {X 0,Y 460.101,Z 625.505,A -85,B 0,C 180,E1 -8010,E2 -8010} C_VEL
LIN {X 0,Y 460.108,Z 625.283,A -85,B 0,C 180,E1 -8010.875,E2 -8010.875} C_VEL
LIN {X 0,Y 459.961,Z 623.61,A -85,B 0,C 180,E1 -8012.627,E2 -8012.627} C_VEL
LIN {X 0,Y 459.976,Z 622.171,A -85,B 0,C 180,E1 -8013.504,E2 -8013.504} C_VEL
LIN {X 0,Y 459.942,Z 619.14,A -85,B 0,C 180,E1 -8014.821,E2 -8014.821} C_VEL
LIN {X 0,Y 459.96,Z 615.048,A -85,B 0,C 180,E1 -8016.14,E2 -8016.14} C_VEL
LIN {X 0,Y 459.919,Z 608.747,A -85,B 0,C 180,E1 -8017.684,E2 -8017.684} C_VEL
LIN {X 0,Y 460.044,Z 601.897,A -85,B 0,C 180,E1 -8019.009,E2 -8019.009} C_VEL
LIN {X 0,Y 460.3,Z 593.427,A -85,B 0,C 180,E1 -8020.335,E2 -8020.335} C_VEL
LIN {X 0,Y 460.611,Z 584.763,A -85,B 0,C 180,E1 -8021.44,E2 -8021.44} C_VEL
LIN {X 0,Y 461.183,Z 574.904,A -85,B 0,C 180,E1 -8022.468,E2 -8022.468} C_VEL
LIN {X 0,Y 461.615,Z 563.588,A -85,B 0,C 180,E1 -8023.425,E2 -8023.425} C_VEL
LIN {X 0,Y 462.194,Z 552.095,A -85,B 0,C 180,E1 -8024.193,E2 -8024.193} C_VEL
LIN {X 0,Y 462.765,Z 540.329,A -85,B 0,C 180,E1 -8024.793,E2 -8024.793} C_VEL
LIN {X 0,Y 463.281,Z 527.731,A -85,B 0,C 180,E1 -8025.254,E2 -8025.254} C_VEL
LIN {X 0,Y 463.609,Z 514.991,A -85,B 0,C 180,E1 -8025.553,E2 -8025.553} C_VEL
LIN {X 0,Y 464.044,Z 434.633,A -85,B 0,C 180,E1 -8026.805,E2 -8026.805} C_VEL
LIN {X 0,Y 461.282,Z 408.981,A -85,B 0,C 180,E1 -8027.332,E2 -8027.332} C_VEL
LIN {X 0,Y 462.039,Z 385.44,A -85,B 0,C 180,E1 -8030.478,E2 -8030.478} C_VEL
LIN {X 0,Y 462.864,Z 364.786,A -85,B 0,C 180,E1 -8033.252,E2 -8033.252} C_VEL
LIN {X 0,Y 463.862,Z 341.634,A -85,B 0,C 180,E1 -8036.385,E2 -8036.385} C_VEL
LIN {X 0,Y 464.268,Z 331.765,A -85,B 0,C 180,E1 -8037.741,E2 -8037.741} C_VEL
LIN {X 0,Y 461.534,Z 318.409,A -85,B 0,C 180,E1 -8039.777,E2 -8039.777} C_VEL
LIN {X 0,Y 460.56,Z 314.215,A -85,B 0,C 180,E1 -8040.489,E2 -8040.489} C_VEL
LIN {X 0,Y 460.514,Z 314.117,A -85,B 0,C 180,E1 -8043.325,E2 -8043.325} C_VEL
LIN {X 0,Y 460.457,Z 314.128,A -85,B 0,C 180,E1 -8046.53,E2 -8046.53} C_VEL
LIN {X 0,Y 460.506,Z 314.113,A -85,B 0,C 180,E1 -8049.864,E2 -8049.864} C_VEL
LIN {X 0,Y 460.458,Z 314.125,A -85,B 0,C 180,E1 -8052.893,E2 -8052.893} C_VEL
LIN {X 0,Y 460.499,Z 314.107,A -85,B 0,C 180,E1 -8055.831,E2 -8055.831} C_VEL
LIN {X 0,Y 460.511,Z 314.119,A -85,B 0,C 180,E1 -8058.986,E2 -8058.986} C_VEL
LIN {X 0,Y 460.477,Z 314.093,A -85,B 0,C 180,E1 -8062.374,E2 -8062.374} C_VEL
LIN {X 0,Y 460.528,Z 314.107,A -85,B 0,C 180,E1 -8065.622,E2 -8065.622} C_VEL
LIN {X 0,Y 460.532,Z 314.115,A -85,B 0,C 180,E1 -8068.744,E2 -8068.744} C_VEL
LIN {X 0,Y 460.543,Z 314.112,A -85,B 0,C 180,E1 -8072.261,E2 -8072.261} C_VEL
LIN {X 0,Y 460.515,Z 314.118,A -85,B 0,C 180,E1 -8074.703,E2 -8074.703} C_VEL
LIN {X 0,Y 460.503,Z 314.119,A -85,B 0,C 180,E1 -8077.571,E2 -8077.571} C_VEL
LIN {X 0,Y 460.56,Z 314.106,A -85,B 0,C 180,E1 -8080.384,E2 -8080.384} C_VEL
LIN {X 0,Y 460.597,Z 314.111,A -85,B 0,C 180,E1 -8084.059,E2 -8084.059} C_VEL
LIN {X 0,Y 460.601,Z 314.104,A -85,B 0,C 180,E1 -8087.666,E2 -8087.666} C_VEL
LIN {X 0,Y 460.603,Z 314.108,A -85,B 0,C 180,E1 -8091.223,E2 -8091.223} C_VEL
LIN {X 0,Y 460.68,Z 314.095,A -85,B 0,C 180,E1 -8093.87,E2 -8093.87} C_VEL
LIN {X 0,Y 460.748,Z 314.092,A -85,B 0,C 180,E1 -8097.377,E2 -8097.377} C_VEL
LIN {X 0,Y 460.809,Z 314.075,A -85,B 0,C 180,E1 -8100,E2 -8100} C_VEL
LIN {X 0,Y 460.758,Z 314.084,A -85,B 0,C 180,E1 -8102.623,E2 -8102.623} C_VEL
LIN {X 0,Y 460.661,Z 314.097,A -85,B 0,C 180,E1 -8106.131,E2 -8106.131} C_VEL
LIN {X 0,Y 460.608,Z 314.099,A -85,B 0,C 180,E1 -8108.777,E2 -8108.777} C_VEL
LIN {X 0,Y 460.589,Z 314.106,A -85,B 0,C 180,E1 -8112.435,E2 -8112.435} C_VEL
LIN {X 0,Y 460.571,Z 314.112,A -85,B 0,C 180,E1 -8115.988,E2 -8115.988} C_VEL
LIN {X 0,Y 460.558,Z 314.113,A -85,B 0,C 180,E1 -8119.616,E2 -8119.616} C_VEL
LIN {X 0,Y 460.5,Z 314.117,A -85,B 0,C 180,E1 -8122.429,E2 -8122.429} C_VEL
LIN {X 0,Y 460.528,Z 314.115,A -85,B 0,C 180,E1 -8125.794,E2 -8125.794} C_VEL
LIN {X 0,Y 460.51,Z 314.098,A -85,B 0,C 180,E1 -8129.233,E2 -8129.233} C_VEL
LIN {X 0,Y 460.518,Z 314.112,A -85,B 0,C 180,E1 -8132.286,E2 -8132.286} C_VEL
LIN {X 0,Y 460.5,Z 314.125,A -85,B 0,C 180,E1 -8135.447,E2 -8135.447} C_VEL
LIN {X 0,Y 460.488,Z 314.108,A -85,B 0,C 180,E1 -8138.89,E2 -8138.89} C_VEL
LIN {X 0,Y 460.497,Z 314.122,A -85,B 0,C 180,E1 -8141.599,E2 -8141.599} C_VEL
LIN {X 0,Y 460.506,Z 314.118,A -85,B 0,C 180,E1 -8144.59,E2 -8144.59} C_VEL
LIN {X 0,Y 460.47,Z 314.122,A -85,B 0,C 180,E1 -8147.814,E2 -8147.814} C_VEL
LIN {X 0,Y 460.507,Z 314.119,A -85,B 0,C 180,E1 -8150.136,E2 -8150.136} C_VEL
LIN {X 0,Y 460.463,Z 314.122,A -85,B 0,C 180,E1 -8153.47,E2 -8153.47} C_VEL
LIN {X 0,Y 460.513,Z 314.117,A -85,B 0,C 180,E1 -8156.675,E2 -8156.675} C_VEL
LIN {X 0,Y 460.492,Z 314.123,A -85,B 0,C 180,E1 -8159.759,E2 -8159.759} C_VEL
LIN {X 0,Y 460.483,Z 314.103,A -85,B 0,C 180,E1 -8162.751,E2 -8162.751} C_VEL
LIN {X 0,Y 460.512,Z 314.123,A -85,B 0,C 180,E1 -8165.667,E2 -8165.667} C_VEL
LIN {X 0,Y 460.522,Z 314.112,A -85,B 0,C 180,E1 -8168.579,E2 -8168.579} C_VEL
LIN {X 0,Y 460.54,Z 314.09,A -85,B 0,C 180,E1 -8171.309,E2 -8171.309} C_VEL
LIN {X 0,Y 460.558,Z 314.248,A -85,B 0,C 180,E1 -8173.003,E2 -8173.003} C_VEL
LIN {X 0,Y 460.785,Z 315.277,A -85,B 0,C 180,E1 -8173.165,E2 -8173.165} C_VEL
LIN {X 0,Y 464.791,Z 326.196,A -85,B 0,C 180,E1 -8173.511,E2 -8173.511} C_VEL
LIN {X 0,Y 464.435,Z 365.486,A -85,B 0,C 180,E1 -8174.12,E2 -8174.12} C_VEL
LIN {X 0,Y 463.81,Z 371.337,A -85,B 0,C 180,E1 -8174.185,E2 -8174.185} C_VEL
LIN {X 0,Y 458.21,Z 390.355,A -85,B 0,C 180,E1 -8174.275,E2 -8174.275} C_VEL
LIN {X 0,Y 457.523,Z 396.164,A -85,B 0,C 180,E1 -8174.374,E2 -8174.374} C_VEL
LIN {X 0,Y 457.387,Z 409.393,A -85,B 0,C 180,E1 -8174.773,E2 -8174.773} C_VEL
LIN {X 0,Y 457.183,Z 421.376,A -85,B 0,C 180,E1 -8175.307,E2 -8175.307} C_VEL
LIN {X 0,Y 456.864,Z 432.626,A -85,B 0,C 180,E1 -8175.977,E2 -8175.977} C_VEL
LIN {X 0,Y 456.301,Z 444.214,A -85,B 0,C 180,E1 -8176.869,E2 -8176.869} C_VEL
LIN {X 0,Y 455.794,Z 454.557,A -85,B 0,C 180,E1 -8177.873,E2 -8177.873} C_VEL
LIN {X 0,Y 455.38,Z 462.987,A -85,B 0,C 180,E1 -8178.877,E2 -8178.877} C_VEL
LIN {X 0,Y 454.901,Z 470.75,A -85,B 0,C 180,E1 -8179.991,E2 -8179.991} C_VEL
LIN {X 0,Y 454.472,Z 478.431,A -85,B 0,C 180,E1 -8181.351,E2 -8181.351} C_VEL
LIN {X 0,Y 454.148,Z 484.189,A -85,B 0,C 180,E1 -8182.619,E2 -8182.619} C_VEL
LIN {X 0,Y 453.969,Z 488.464,A -85,B 0,C 180,E1 -8183.779,E2 -8183.779} C_VEL
LIN {X 0,Y 453.626,Z 492.359,A -85,B 0,C 180,E1 -8185.112,E2 -8185.112} C_VEL
LIN {X 0,Y 453.405,Z 495.229,A -85,B 0,C 180,E1 -8186.445,E2 -8186.445} C_VEL
LIN {X 0,Y 453.446,Z 496.587,A -85,B 0,C 180,E1 -8187.335,E2 -8187.335} C_VEL
LIN {X 0,Y 453.313,Z 497.573,A -85,B 0,C 180,E1 -8188.223,E2 -8188.223} C_VEL
LIN {X 0,Y 453.392,Z 498.159,A -85,B 0,C 180,E1 -8189.112,E2 -8189.112} C_VEL
LIN {X 0,Y 453.376,Z 498.39,A -85,B 0,C 180,E1 -8190,E2 -8190} C_VEL
LIN {X 0,Y 453.392,Z 498.207,A -85,B 0,C 180,E1 -8190.888,E2 -8190.888} C_VEL
LIN {X 0,Y 453.313,Z 497.652,A -85,B 0,C 180,E1 -8191.777,E2 -8191.777} C_VEL
LIN {X 0,Y 453.445,Z 496.697,A -85,B 0,C 180,E1 -8192.665,E2 -8192.665} C_VEL
LIN {X 0,Y 453.398,Z 495.39,A -85,B 0,C 180,E1 -8193.555,E2 -8193.555} C_VEL
LIN {X 0,Y 453.62,Z 492.58,A -85,B 0,C 180,E1 -8194.888,E2 -8194.888} C_VEL
LIN {X 0,Y 453.955,Z 488.76,A -85,B 0,C 180,E1 -8196.221,E2 -8196.221} C_VEL
LIN {X 0,Y 454.126,Z 483.685,A -85,B 0,C 180,E1 -8197.604,E2 -8197.604} C_VEL
LIN {X 0,Y 454.629,Z 476.458,A -85,B 0,C 180,E1 -8199.117,E2 -8199.117} C_VEL
LIN {X 0,Y 455.144,Z 468.434,A -85,B 0,C 180,E1 -8200.453,E2 -8200.453} C_VEL
LIN {X 0,Y 455.56,Z 460.216,A -85,B 0,C 180,E1 -8201.569,E2 -8201.569} C_VEL
LIN {X 0,Y 456.021,Z 451.191,A -85,B 0,C 180,E1 -8202.573,E2 -8202.573} C_VEL
LIN {X 0,Y 456.578,Z 440.7,A -85,B 0,C 180,E1 -8203.514,E2 -8203.514} C_VEL
LIN {X 0,Y 456.938,Z 429.206,A -85,B 0,C 180,E1 -8204.338,E2 -8204.338} C_VEL
LIN {X 0,Y 457.221,Z 417.973,A -85,B 0,C 180,E1 -8204.959,E2 -8204.959} C_VEL
LIN {X 0,Y 457.437,Z 404.803,A -85,B 0,C 180,E1 -8205.482,E2 -8205.482} C_VEL
LIN {X 0,Y 457.463,Z 391.09,A -85,B 0,C 180,E1 -8205.824,E2 -8205.824} C_VEL
LIN {X 0,Y 457.889,Z 327.208,A -85,B 0,C 180,E1 -8206.839,E2 -8206.839} C_VEL
LIN {X 0,Y 453.66,Z 315.921,A -85,B 0,C 180,E1 -8207.219,E2 -8207.219} C_VEL
LIN {X 0,Y 453.51,Z 315.152,A -85,B 0,C 180,E1 -8207.356,E2 -8207.356} C_VEL
LIN {X 0,Y 453.482,Z 314.996,A -85,B 0,C 180,E1 -8209.935,E2 -8209.935} C_VEL
LIN {X 0,Y 453.476,Z 314.985,A -85,B 0,C 180,E1 -8212.796,E2 -8212.796} C_VEL
LIN {X 0,Y 453.465,Z 314.992,A -85,B 0,C 180,E1 -8215.984,E2 -8215.984} C_VEL
LIN {X 0,Y 453.458,Z 314.986,A -85,B 0,C 180,E1 -8218.715,E2 -8218.715} C_VEL
LIN {X 0,Y 453.433,Z 314.999,A -85,B 0,C 180,E1 -8221.801,E2 -8221.801} C_VEL
LIN {X 0,Y 453.469,Z 315,A -85,B 0,C 180,E1 -8224.99,E2 -8224.99} C_VEL
LIN {X 0,Y 453.447,Z 314.993,A -85,B 0,C 180,E1 -8228.313,E2 -8228.313} C_VEL
LIN {X 0,Y 453.467,Z 315.002,A -85,B 0,C 180,E1 -8230.611,E2 -8230.611} C_VEL
LIN {X 0,Y 453.477,Z 314.989,A -85,B 0,C 180,E1 -8234.528,E2 -8234.528} C_VEL
LIN {X 0,Y 453.43,Z 315.002,A -85,B 0,C 180,E1 -8238.071,E2 -8238.071} C_VEL
LIN {X 0,Y 453.434,Z 314.985,A -85,B 0,C 180,E1 -8240.801,E2 -8240.801} C_VEL
LIN {X 0,Y 453.443,Z 314.996,A -85,B 0,C 180,E1 -8243.916,E2 -8243.916} C_VEL
LIN {X 0,Y 453.468,Z 314.991,A -85,B 0,C 180,E1 -8247.15,E2 -8247.15} C_VEL
LIN {X 0,Y 453.45,Z 314.976,A -85,B 0,C 180,E1 -8250.266,E2 -8250.266} C_VEL
LIN {X 0,Y 453.435,Z 314.994,A -85,B 0,C 180,E1 -8253.289,E2 -8253.289} C_VEL
LIN {X 0,Y 453.474,Z 314.999,A -85,B 0,C 180,E1 -8256.237,E2 -8256.237} C_VEL
LIN {X 0,Y 453.463,Z 314.99,A -85,B 0,C 180,E1 -8259.117,E2 -8259.117} C_VEL
LIN {X 0,Y 453.485,Z 314.994,A -85,B 0,C 180,E1 -8261.943,E2 -8261.943} C_VEL
LIN {X 0,Y 453.521,Z 314.983,A -85,B 0,C 180,E1 -8264.726,E2 -8264.726} C_VEL
LIN {X 0,Y 453.548,Z 314.991,A -85,B 0,C 180,E1 -8268.379,E2 -8268.379} C_VEL
LIN {X 0,Y 453.552,Z 314.979,A -85,B 0,C 180,E1 -8271.086,E2 -8271.086} C_VEL
LIN {X 0,Y 453.619,Z 314.973,A -85,B 0,C 180,E1 -8273.774,E2 -8273.774} C_VEL
LIN {X 0,Y 453.705,Z 314.963,A -85,B 0,C 180,E1 -8277.336,E2 -8277.336} C_VEL
LIN {X 0,Y 453.738,Z 314.955,A -85,B 0,C 180,E1 -8280,E2 -8280} C_VEL
LIN {X 0,Y 453.694,Z 314.97,A -85,B 0,C 180,E1 -8282.664,E2 -8282.664} C_VEL
LIN {X 0,Y 453.647,Z 314.969,A -85,B 0,C 180,E1 -8286.226,E2 -8286.226} C_VEL
LIN {X 0,Y 453.563,Z 314.984,A -85,B 0,C 180,E1 -8288.914,E2 -8288.914} C_VEL
LIN {X 0,Y 453.557,Z 314.98,A -85,B 0,C 180,E1 -8292.529,E2 -8292.529} C_VEL
LIN {X 0,Y 453.537,Z 314.994,A -85,B 0,C 180,E1 -8296.196,E2 -8296.196} C_VEL
LIN {X 0,Y 453.51,Z 314.982,A -85,B 0,C 180,E1 -8299.039,E2 -8299.039} C_VEL
LIN {X 0,Y 453.47,Z 314.985,A -85,B 0,C 180,E1 -8301.837,E2 -8301.837} C_VEL
LIN {X 0,Y 453.462,Z 314.998,A -85,B 0,C 180,E1 -8304.737,E2 -8304.737} C_VEL
LIN {X 0,Y 453.483,Z 314.989,A -85,B 0,C 180,E1 -8307.95,E2 -8307.95} C_VEL
LIN {X 0,Y 453.469,Z 314.997,A -85,B 0,C 180,E1 -8310.76,E2 -8310.76} C_VEL
LIN {X 0,Y 453.459,Z 314.996,A -85,B 0,C 180,E1 -8313.914,E2 -8313.914} C_VEL
LIN {X 0,Y 453.429,Z 315.001,A -85,B 0,C 180,E1 -8317.192,E2 -8317.192} C_VEL
LIN {X 0,Y 453.465,Z 314.998,A -85,B 0,C 180,E1 -8320.612,E2 -8320.612} C_VEL
LIN {X 0,Y 453.454,Z 314.983,A -85,B 0,C 180,E1 -8324.223,E2 -8324.223} C_VEL
LIN {X 0,Y 453.413,Z 315.002,A -85,B 0,C 180,E1 -8327,E2 -8327} C_VEL
LIN {X 0,Y 453.467,Z 314.995,A -85,B 0,C 180,E1 -8329.413,E2 -8329.413} C_VEL
LIN {X 0,Y 453.432,Z 315.002,A -85,B 0,C 180,E1 -8332.809,E2 -8332.809} C_VEL
LIN {X 0,Y 453.463,Z 315,A -85,B 0,C 180,E1 -8336.087,E2 -8336.087} C_VEL
LIN {X 0,Y 453.537,Z 315.14,A -85,B 0,C 180,E1 -8339.272,E2 -8339.272} C_VEL
LIN {X 0,Y 456.658,Z 329.075,A -85,B 0,C 180,E1 -8341.505,E2 -8341.505} C_VEL
LIN {X 0,Y 457.342,Z 332.657,A -85,B 0,C 180,E1 -8342.051,E2 -8342.051} C_VEL
LIN {X 0,Y 456.727,Z 348.294,A -85,B 0,C 180,E1 -8344.234,E2 -8344.234} C_VEL
LIN {X 0,Y 455.568,Z 374.004,A -85,B 0,C 180,E1 -8347.761,E2 -8347.761} C_VEL
LIN {X 0,Y 454.555,Z 399.791,A -85,B 0,C 180,E1 -8351.288,E2 -8351.288} C_VEL
LIN {X 0,Y 454.273,Z 408.127,A -85,B 0,C 180,E1 -8352.398,E2 -8352.398} C_VEL
LIN {X 0,Y 457.337,Z 437.201,A -85,B 0,C 180,E1 -8352.995,E2 -8352.995} C_VEL
LIN {X 0,Y 456.683,Z 518.464,A -85,B 0,C 180,E1 -8354.291,E2 -8354.291} C_VEL
LIN {X 0,Y 456.185,Z 531.782,A -85,B 0,C 180,E1 -8354.674,E2 -8354.674} C_VEL
LIN {X 0,Y 455.606,Z 544.016,A -85,B 0,C 180,E1 -8355.198,E2 -8355.198} C_VEL
LIN {X 0,Y 455.007,Z 556.408,A -85,B 0,C 180,E1 -8355.92,E2 -8355.92} C_VEL
LIN {X 0,Y 454.446,Z 567.78,A -85,B 0,C 180,E1 -8356.783,E2 -8356.783} C_VEL
LIN {X 0,Y 453.983,Z 578.759,A -85,B 0,C 180,E1 -8357.824,E2 -8357.824} C_VEL
LIN {X 0,Y 453.479,Z 587.437,A -85,B 0,C 180,E1 -8358.83,E2 -8358.83} C_VEL
LIN {X 0,Y 453.133,Z 595.479,A -85,B 0,C 180,E1 -8359.951,E2 -8359.951} C_VEL
LIN {X 0,Y 452.933,Z 603.369,A -85,B 0,C 180,E1 -8361.299,E2 -8361.299} C_VEL
LIN {X 0,Y 452.82,Z 610.659,A -85,B 0,C 180,E1 -8362.868,E2 -8362.868} C_VEL
LIN {X 0,Y 452.848,Z 615.531,A -85,B 0,C 180,E1 -8364.21,E2 -8364.21} C_VEL
LIN {X 0,Y 452.911,Z 619.263,A -85,B 0,C 180,E1 -8365.55,E2 -8365.55} C_VEL
LIN {X 0,Y 452.929,Z 621.186,A -85,B 0,C 180,E1 -8366.442,E2 -8366.442} C_VEL
LIN {X 0,Y 452.916,Z 622.626,A -85,B 0,C 180,E1 -8367.332,E2 -8367.332} C_VEL
LIN {X 0,Y 453.084,Z 624.305,A -85,B 0,C 180,E1 -8369.111,E2 -8369.111} C_VEL
LIN {X 0,Y 453.079,Z 624.527,A -85,B 0,C 180,E1 -8370,E2 -8370} C_VEL
LIN {X 0,Y 453.084,Z 624.305,A -85,B 0,C 180,E1 -8370.889,E2 -8370.889} C_VEL
LIN {X 0,Y 452.916,Z 622.628,A -85,B 0,C 180,E1 -8372.668,E2 -8372.668} C_VEL
LIN {X 0,Y 452.929,Z 621.188,A -85,B 0,C 180,E1 -8373.558,E2 -8373.558} C_VEL
LIN {X 0,Y 452.886,Z 618.154,A -85,B 0,C 180,E1 -8374.896,E2 -8374.896} C_VEL
LIN {X 0,Y 452.88,Z 614.056,A -85,B 0,C 180,E1 -8376.236,E2 -8376.236} C_VEL
LIN {X 0,Y 452.862,Z 607.755,A -85,B 0,C 180,E1 -8377.804,E2 -8377.804} C_VEL
LIN {X 0,Y 452.995,Z 600.903,A -85,B 0,C 180,E1 -8379.15,E2 -8379.15} C_VEL
LIN {X 0,Y 453.27,Z 592.43,A -85,B 0,C 180,E1 -8380.497,E2 -8380.497} C_VEL
LIN {X 0,Y 453.588,Z 583.763,A -85,B 0,C 180,E1 -8381.62,E2 -8381.62} C_VEL
LIN {X 0,Y 454.141,Z 574.49,A -85,B 0,C 180,E1 -8382.609,E2 -8382.609} C_VEL
LIN {X 0,Y 454.631,Z 562.585,A -85,B 0,C 180,E1 -8383.635,E2 -8383.635} C_VEL
LIN {X 0,Y 455.307,Z 551.102,A -85,B 0,C 180,E1 -8384.412,E2 -8384.412} C_VEL
LIN {X 0,Y 455.87,Z 539.33,A -85,B 0,C 180,E1 -8385.022,E2 -8385.022} C_VEL
LIN {X 0,Y 456.434,Z 526.734,A -85,B 0,C 180,E1 -8385.489,E2 -8385.489} C_VEL
LIN {X 0,Y 456.788,Z 513.991,A -85,B 0,C 180,E1 -8385.791,E2 -8385.791} C_VEL
LIN {X 0,Y 457.171,Z 434.639,A -85,B 0,C 180,E1 -8387.049,E2 -8387.049} C_VEL
LIN {X 0,Y 454.262,Z 408.06,A -85,B 0,C 180,E1 -8387.603,E2 -8387.603} C_VEL
LIN {X 0,Y 455.028,Z 386.194,A -85,B 0,C 180,E1 -8390.571,E2 -8390.571} C_VEL
LIN {X 0,Y 455.894,Z 365.584,A -85,B 0,C 180,E1 -8393.388,E2 -8393.388} C_VEL
LIN {X 0,Y 456.881,Z 344.791,A -85,B 0,C 180,E1 -8396.247,E2 -8396.247} C_VEL
LIN {X 0,Y 457.303,Z 332.616,A -85,B 0,C 180,E1 -8397.952,E2 -8397.952} C_VEL
LIN {X 0,Y 454.117,Z 317.655,A -85,B 0,C 180,E1 -8400.286,E2 -8400.286} C_VEL
LIN {X 0,Y 453.502,Z 315.085,A -85,B 0,C 180,E1 -8400.757,E2 -8400.757} C_VEL
LIN {X 0,Y 453.463,Z 315.001,A -85,B 0,C 180,E1 -8403.913,E2 -8403.913} C_VEL
LIN {X 0,Y 453.433,Z 315.002,A -85,B 0,C 180,E1 -8407.191,E2 -8407.191} C_VEL
LIN {X 0,Y 453.466,Z 314.996,A -85,B 0,C 180,E1 -8410.611,E2 -8410.611} C_VEL
LIN {X 0,Y 453.477,Z 314.977,A -85,B 0,C 180,E1 -8414.528,E2 -8414.528} C_VEL
LIN {X 0,Y 453.435,Z 315.007,A -85,B 0,C 180,E1 -8418.07,E2 -8418.07} C_VEL
LIN {X 0,Y 453.433,Z 314.991,A -85,B 0,C 180,E1 -8420.802,E2 -8420.802} C_VEL
LIN {X 0,Y 453.436,Z 314.974,A -85,B 0,C 180,E1 -8423.915,E2 -8423.915} C_VEL
LIN {X 0,Y 453.468,Z 314.994,A -85,B 0,C 180,E1 -8427.15,E2 -8427.15} C_VEL
LIN {X 0,Y 453.461,Z 314.991,A -85,B 0,C 180,E1 -8430.267,E2 -8430.267} C_VEL
LIN {X 0,Y 453.455,Z 314.993,A -85,B 0,C 180,E1 -8433.291,E2 -8433.291} C_VEL
LIN {X 0,Y 453.485,Z 314.993,A -85,B 0,C 180,E1 -8436.238,E2 -8436.238} C_VEL
LIN {X 0,Y 453.474,Z 314.981,A -85,B 0,C 180,E1 -8439.117,E2 -8439.117} C_VEL
LIN {X 0,Y 453.494,Z 314.995,A -85,B 0,C 180,E1 -8441.944,E2 -8441.944} C_VEL
LIN {X 0,Y 453.531,Z 314.987,A -85,B 0,C 180,E1 -8444.726,E2 -8444.726} C_VEL
LIN {X 0,Y 453.549,Z 314.984,A -85,B 0,C 180,E1 -8448.379,E2 -8448.379} C_VEL
LIN {X 0,Y 453.57,Z 314.983,A -85,B 0,C 180,E1 -8451.086,E2 -8451.086} C_VEL
LIN {X 0,Y 453.647,Z 314.97,A -85,B 0,C 180,E1 -8453.774,E2 -8453.774} C_VEL
LIN {X 0,Y 453.695,Z 314.97,A -85,B 0,C 180,E1 -8457.336,E2 -8457.336} C_VEL
LIN {X 0,Y 453.758,Z 314.953,A -85,B 0,C 180,E1 -8460,E2 -8460} C_VEL
LIN {X 0,Y 453.706,Z 314.963,A -85,B 0,C 180,E1 -8462.664,E2 -8462.664} C_VEL
LIN {X 0,Y 453.629,Z 314.972,A -85,B 0,C 180,E1 -8466.226,E2 -8466.226} C_VEL
LIN {X 0,Y 453.575,Z 314.976,A -85,B 0,C 180,E1 -8468.914,E2 -8468.914} C_VEL
LIN {X 0,Y 453.557,Z 314.982,A -85,B 0,C 180,E1 -8472.529,E2 -8472.529} C_VEL
LIN {X 0,Y 453.53,Z 314.987,A -85,B 0,C 180,E1 -8476.197,E2 -8476.197} C_VEL
LIN {X 0,Y 453.51,Z 314.991,A -85,B 0,C 180,E1 -8479.04,E2 -8479.04} C_VEL
LIN {X 0,Y 453.469,Z 314.998,A -85,B 0,C 180,E1 -8481.837,E2 -8481.837} C_VEL
LIN {X 0,Y 453.462,Z 314.996,A -85,B 0,C 180,E1 -8484.738,E2 -8484.738} C_VEL
LIN {X 0,Y 453.455,Z 314.98,A -85,B 0,C 180,E1 -8487.943,E2 -8487.943} C_VEL
LIN {X 0,Y 453.449,Z 314.978,A -85,B 0,C 180,E1 -8490.762,E2 -8490.762} C_VEL
LIN {X 0,Y 453.461,Z 314.999,A -85,B 0,C 180,E1 -8493.914,E2 -8493.914} C_VEL
LIN {X 0,Y 453.441,Z 314.998,A -85,B 0,C 180,E1 -8497.191,E2 -8497.191} C_VEL
LIN {X 0,Y 453.465,Z 314.986,A -85,B 0,C 180,E1 -8500.612,E2 -8500.612} C_VEL
LIN {X 0,Y 453.476,Z 314.993,A -85,B 0,C 180,E1 -8504.529,E2 -8504.529} C_VEL
LIN {X 0,Y 453.432,Z 314.997,A -85,B 0,C 180,E1 -8508.072,E2 -8508.072} C_VEL
LIN {X 0,Y 453.44,Z 315.001,A -85,B 0,C 180,E1 -8510.802,E2 -8510.802} C_VEL
LIN {X 0,Y 453.445,Z 314.999,A -85,B 0,C 180,E1 -8513.917,E2 -8513.917} C_VEL
LIN {X 0,Y 453.469,Z 314.994,A -85,B 0,C 180,E1 -8517.151,E2 -8517.151} C_VEL
LIN {X 0,Y 453.453,Z 314.997,A -85,B 0,C 180,E1 -8520.267,E2 -8520.267} C_VEL
LIN {X 0,Y 453.422,Z 314.985,A -85,B 0,C 180,E1 -8523.289,E2 -8523.289} C_VEL
LIN {X 0,Y 453.49,Z 314.995,A -85,B 0,C 180,E1 -8526.239,E2 -8526.239} C_VEL
LIN {X 0,Y 453.482,Z 314.995,A -85,B 0,C 180,E1 -8529.118,E2 -8529.118} C_VEL
LIN {X 0,Y 453.473,Z 314.953,A -85,B 0,C 180,E1 -8531.943,E2 -8531.943} C_VEL
LIN {X 0,Y 453.537,Z 315.212,A -85,B 0,C 180,E1 -8532.761,E2 -8532.761} C_VEL
LIN {X 0,Y 453.811,Z 316.32,A -85,B 0,C 180,E1 -8532.902,E2 -8532.902} C_VEL
LIN {X 0,Y 458.001,Z 327.943,A -85,B 0,C 180,E1 -8533.272,E2 -8533.272} C_VEL
LIN {X 0,Y 457.523,Z 396.164,A -85,B 0,C 180,E1 -8534.374,E2 -8534.374} C_VEL
LIN {X 0,Y 456.844,Z 401.951,A -85,B 0,C 180,E1 -8534.499,E2 -8534.499} C_VEL
LIN {X 0,Y 454.032,Z 411.309,A -85,B 0,C 180,E1 -8534.709,E2 -8534.709} C_VEL
LIN {X 0,Y 451.107,Z 420.451,A -85,B 0,C 180,E1 -8535.009,E2 -8535.009} C_VEL
LIN {X 0,Y 450.27,Z 425.89,A -85,B 0,C 180,E1 -8535.276,E2 -8535.276} C_VEL
LIN {X 0,Y 449.979,Z 436.645,A -85,B 0,C 180,E1 -8535.982,E2 -8535.982} C_VEL
LIN {X 0,Y 449.394,Z 446.468,A -85,B 0,C 180,E1 -8536.779,E2 -8536.779} C_VEL
LIN {X 0,Y 448.874,Z 456.586,A -85,B 0,C 180,E1 -8537.798,E2 -8537.798} C_VEL
LIN {X 0,Y 448.412,Z 465.642,A -85,B 0,C 180,E1 -8538.931,E2 -8538.931} C_VEL
LIN {X 0,Y 447.832,Z 474.424,A -85,B 0,C 180,E1 -8540.288,E2 -8540.288} C_VEL
LIN {X 0,Y 447.454,Z 480.607,A -85,B 0,C 180,E1 -8541.464,E2 -8541.464} C_VEL
LIN {X 0,Y 447.146,Z 486.224,A -85,B 0,C 180,E1 -8542.777,E2 -8542.777} C_VEL
LIN {X 0,Y 446.778,Z 490.848,A -85,B 0,C 180,E1 -8544.132,E2 -8544.132} C_VEL
LIN {X 0,Y 446.519,Z 494.383,A -85,B 0,C 180,E1 -8545.486,E2 -8545.486} C_VEL
LIN {X 0,Y 446.386,Z 496.209,A -85,B 0,C 180,E1 -8546.389,E2 -8546.389} C_VEL
LIN {X 0,Y 446.428,Z 497.565,A -85,B 0,C 180,E1 -8547.293,E2 -8547.293} C_VEL
LIN {X 0,Y 446.291,Z 498.551,A -85,B 0,C 180,E1 -8548.195,E2 -8548.195} C_VEL
LIN {X 0,Y 446.371,Z 499.136,A -85,B 0,C 180,E1 -8549.098,E2 -8549.098} C_VEL
LIN {X 0,Y 446.354,Z 499.367,A -85,B 0,C 180,E1 -8550,E2 -8550} C_VEL
LIN {X 0,Y 446.37,Z 499.184,A -85,B 0,C 180,E1 -8550.902,E2 -8550.902} C_VEL
LIN {X 0,Y 446.291,Z 498.629,A -85,B 0,C 180,E1 -8551.805,E2 -8551.805} C_VEL
LIN {X 0,Y 446.426,Z 497.674,A -85,B 0,C 180,E1 -8552.707,E2 -8552.707} C_VEL
LIN {X 0,Y 446.38,Z 496.368,A -85,B 0,C 180,E1 -8553.611,E2 -8553.611} C_VEL
LIN {X 0,Y 446.615,Z 493.557,A -85,B 0,C 180,E1 -8554.965,E2 -8554.965} C_VEL
LIN {X 0,Y 446.971,Z 489.737,A -85,B 0,C 180,E1 -8556.319,E2 -8556.319} C_VEL
LIN {X 0,Y 447.161,Z 484.661,A -85,B 0,C 180,E1 -8557.723,E2 -8557.723} C_VEL
LIN {X 0,Y 447.692,Z 477.434,A -85,B 0,C 180,E1 -8559.259,E2 -8559.259} C_VEL
LIN {X 0,Y 448.237,Z 469.409,A -85,B 0,C 180,E1 -8560.616,E2 -8560.616} C_VEL
LIN {X 0,Y 448.675,Z 461.191,A -85,B 0,C 180,E1 -8561.749,E2 -8561.749} C_VEL
LIN {X 0,Y 449.164,Z 452.165,A -85,B 0,C 180,E1 -8562.768,E2 -8562.768} C_VEL
LIN {X 0,Y 449.747,Z 441.672,A -85,B 0,C 180,E1 -8563.723,E2 -8563.723} C_VEL
LIN {X 0,Y 450.133,Z 430.023,A -85,B 0,C 180,E1 -8564.57,E2 -8564.57} C_VEL
LIN {X 0,Y 450.45,Z 418.607,A -85,B 0,C 180,E1 -8565.207,E2 -8565.207} C_VEL
LIN {X 0,Y 450.652,Z 405.769,A -85,B 0,C 180,E1 -8565.721,E2 -8565.721} C_VEL
LIN {X 0,Y 450.676,Z 392.049,A -85,B 0,C 180,E1 -8566.069,E2 -8566.069} C_VEL
LIN {X 0,Y 451.187,Z 329.465,A -85,B 0,C 180,E1 -8567.075,E2 -8567.075} C_VEL
LIN {X 0,Y 447.226,Z 318.418,A -85,B 0,C 180,E1 -8567.424,E2 -8567.424} C_VEL
LIN {X 0,Y 446.564,Z 316.407,A -85,B 0,C 180,E1 -8567.546,E2 -8567.546} C_VEL
LIN {X 0,Y 446.452,Z 315.875,A -85,B 0,C 180,E1 -8567.758,E2 -8567.758} C_VEL
LIN {X 0,Y 446.428,Z 315.876,A -85,B 0,C 180,E1 -8570.263,E2 -8570.263} C_VEL
LIN {X 0,Y 446.421,Z 315.867,A -85,B 0,C 180,E1 -8573.177,E2 -8573.177} C_VEL
LIN {X 0,Y 446.416,Z 315.865,A -85,B 0,C 180,E1 -8576.186,E2 -8576.186} C_VEL
LIN {X 0,Y 446.415,Z 315.872,A -85,B 0,C 180,E1 -8579.211,E2 -8579.211} C_VEL
LIN {X 0,Y 446.395,Z 315.875,A -85,B 0,C 180,E1 -8582.363,E2 -8582.363} C_VEL
LIN {X 0,Y 446.41,Z 315.875,A -85,B 0,C 180,E1 -8585.626,E2 -8585.626} C_VEL
LIN {X 0,Y 446.4,Z 315.88,A -85,B 0,C 180,E1 -8589.031,E2 -8589.031} C_VEL
LIN {X 0,Y 446.376,Z 315.876,A -85,B 0,C 180,E1 -8592.269,E2 -8592.269} C_VEL
LIN {X 0,Y 446.445,Z 315.872,A -85,B 0,C 180,E1 -8595.104,E2 -8595.104} C_VEL
LIN {X 0,Y 446.395,Z 315.875,A -85,B 0,C 180,E1 -8598.605,E2 -8598.605} C_VEL
LIN {X 0,Y 446.399,Z 315.861,A -85,B 0,C 180,E1 -8601.922,E2 -8601.922} C_VEL
LIN {X 0,Y 446.415,Z 315.874,A -85,B 0,C 180,E1 -8605.476,E2 -8605.476} C_VEL
LIN {X 0,Y 446.402,Z 315.861,A -85,B 0,C 180,E1 -8608.698,E2 -8608.698} C_VEL
LIN {X 0,Y 446.417,Z 315.854,A -85,B 0,C 180,E1 -8611.836,E2 -8611.836} C_VEL
LIN {X 0,Y 446.414,Z 315.878,A -85,B 0,C 180,E1 -8614.845,E2 -8614.845} C_VEL
LIN {X 0,Y 446.438,Z 315.872,A -85,B 0,C 180,E1 -8618.246,E2 -8618.246} C_VEL
LIN {X 0,Y 446.437,Z 315.871,A -85,B 0,C 180,E1 -8621.648,E2 -8621.648} C_VEL
LIN {X 0,Y 446.484,Z 315.863,A -85,B 0,C 180,E1 -8624.479,E2 -8624.479} C_VEL
LIN {X 0,Y 446.507,Z 315.865,A -85,B 0,C 180,E1 -8628.193,E2 -8628.193} C_VEL
LIN {X 0,Y 446.503,Z 315.858,A -85,B 0,C 180,E1 -8630.944,E2 -8630.944} C_VEL
LIN {X 0,Y 446.59,Z 315.848,A -85,B 0,C 180,E1 -8633.675,E2 -8633.675} C_VEL
LIN {X 0,Y 446.655,Z 315.841,A -85,B 0,C 180,E1 -8637.294,E2 -8637.294} C_VEL
LIN {X 0,Y 446.689,Z 315.833,A -85,B 0,C 180,E1 -8640,E2 -8640} C_VEL
LIN {X 0,Y 446.643,Z 315.848,A -85,B 0,C 180,E1 -8642.706,E2 -8642.706} C_VEL
LIN {X 0,Y 446.616,Z 315.845,A -85,B 0,C 180,E1 -8646.324,E2 -8646.324} C_VEL
LIN {X 0,Y 446.511,Z 315.862,A -85,B 0,C 180,E1 -8649.056,E2 -8649.056} C_VEL
LIN {X 0,Y 446.514,Z 315.856,A -85,B 0,C 180,E1 -8652.73,E2 -8652.73} C_VEL
LIN {X 0,Y 446.48,Z 315.87,A -85,B 0,C 180,E1 -8656.459,E2 -8656.459} C_VEL
LIN {X 0,Y 446.461,Z 315.859,A -85,B 0,C 180,E1 -8659.304,E2 -8659.304} C_VEL
LIN {X 0,Y 446.411,Z 315.869,A -85,B 0,C 180,E1 -8662.2,E2 -8662.2} C_VEL
LIN {X 0,Y 446.414,Z 315.874,A -85,B 0,C 180,E1 -8665.155,E2 -8665.155} C_VEL
LIN {X 0,Y 446.434,Z 315.865,A -85,B 0,C 180,E1 -8668.182,E2 -8668.182} C_VEL
LIN {X 0,Y 446.408,Z 315.875,A -85,B 0,C 180,E1 -8671.301,E2 -8671.301} C_VEL
LIN {X 0,Y 446.414,Z 315.87,A -85,B 0,C 180,E1 -8674.524,E2 -8674.524} C_VEL
LIN {X 0,Y 446.392,Z 315.88,A -85,B 0,C 180,E1 -8678.077,E2 -8678.077} C_VEL
LIN {X 0,Y 446.397,Z 315.878,A -85,B 0,C 180,E1 -8681.395,E2 -8681.395} C_VEL
LIN {X 0,Y 446.415,Z 315.854,A -85,B 0,C 180,E1 -8684.893,E2 -8684.893} C_VEL
LIN {X 0,Y 446.396,Z 315.876,A -85,B 0,C 180,E1 -8688.606,E2 -8688.606} C_VEL
LIN {X 0,Y 446.395,Z 315.879,A -85,B 0,C 180,E1 -8691.924,E2 -8691.924} C_VEL
LIN {X 0,Y 446.417,Z 315.876,A -85,B 0,C 180,E1 -8695.477,E2 -8695.477} C_VEL
LIN {X 0,Y 446.492,Z 316.014,A -85,B 0,C 180,E1 -8699.003,E2 -8699.003} C_VEL
LIN {X 0,Y 449.673,Z 330.192,A -85,B 0,C 180,E1 -8701.317,E2 -8701.317} C_VEL
LIN {X 0,Y 450.494,Z 335.261,A -85,B 0,C 180,E1 -8702.095,E2 -8702.095} C_VEL
LIN {X 0,Y 449.347,Z 358.426,A -85,B 0,C 180,E1 -8705.36,E2 -8705.36} C_VEL
LIN {X 0,Y 448.338,Z 380.145,A -85,B 0,C 180,E1 -8708.385,E2 -8708.385} C_VEL
LIN {X 0,Y 447.319,Z 405.672,A -85,B 0,C 180,E1 -8711.947,E2 -8711.947} C_VEL
LIN {X 0,Y 447.327,Z 407.367,A -85,B 0,C 180,E1 -8712.125,E2 -8712.125} C_VEL
LIN {X 0,Y 450.505,Z 438.018,A -85,B 0,C 180,E1 -8712.758,E2 -8712.758} C_VEL
LIN {X 0,Y 449.83,Z 517.484,A -85,B 0,C 180,E1 -8714.045,E2 -8714.045} C_VEL
LIN {X 0,Y 449.338,Z 530.801,A -85,B 0,C 180,E1 -8714.435,E2 -8714.435} C_VEL
LIN {X 0,Y 448.66,Z 544.16,A -85,B 0,C 180,E1 -8715.021,E2 -8715.021} C_VEL
LIN {X 0,Y 448.074,Z 555.417,A -85,B 0,C 180,E1 -8715.698,E2 -8715.698} C_VEL
LIN {X 0,Y 447.42,Z 567.138,A -85,B 0,C 180,E1 -8716.603,E2 -8716.603} C_VEL
LIN {X 0,Y 446.999,Z 577.767,A -85,B 0,C 180,E1 -8717.63,E2 -8717.63} C_VEL
LIN {X 0,Y 446.436,Z 586.44,A -85,B 0,C 180,E1 -8718.651,E2 -8718.651} C_VEL
LIN {X 0,Y 446.1,Z 594.486,A -85,B 0,C 180,E1 -8719.791,E2 -8719.791} C_VEL
LIN {X 0,Y 445.846,Z 602.372,A -85,B 0,C 180,E1 -8721.159,E2 -8721.159} C_VEL
LIN {X 0,Y 445.779,Z 607.795,A -85,B 0,C 180,E1 -8722.299,E2 -8722.299} C_VEL
LIN {X 0,Y 445.779,Z 613.067,A -85,B 0,C 180,E1 -8723.664,E2 -8723.664} C_VEL
LIN {X 0,Y 445.83,Z 617.17,A -85,B 0,C 180,E1 -8725.026,E2 -8725.026} C_VEL
LIN {X 0,Y 445.884,Z 620.204,A -85,B 0,C 180,E1 -8726.385,E2 -8726.385} C_VEL
LIN {X 0,Y 445.87,Z 621.645,A -85,B 0,C 180,E1 -8727.29,E2 -8727.29} C_VEL
LIN {X 0,Y 446.058,Z 623.327,A -85,B 0,C 180,E1 -8729.097,E2 -8729.097} C_VEL
LIN {X 0,Y 446.056,Z 623.55,A -85,B 0,C 180,E1 -8730,E2 -8730} C_VEL
LIN {X 0,Y 446.058,Z 623.327,A -85,B 0,C 180,E1 -8730.903,E2 -8730.903} C_VEL
LIN {X 0,Y 445.871,Z 621.647,A -85,B 0,C 180,E1 -8732.71,E2 -8732.71} C_VEL
LIN {X 0,Y 445.884,Z 620.206,A -85,B 0,C 180,E1 -8733.615,E2 -8733.615} C_VEL
LIN {X 0,Y 445.832,Z 617.168,A -85,B 0,C 180,E1 -8734.974,E2 -8734.974} C_VEL
LIN {X 0,Y 445.807,Z 613.065,A -85,B 0,C 180,E1 -8736.336,E2 -8736.336} C_VEL
LIN {X 0,Y 445.801,Z 606.762,A -85,B 0,C 180,E1 -8737.929,E2 -8737.929} C_VEL
LIN {X 0,Y 445.92,Z 599.904,A -85,B 0,C 180,E1 -8739.296,E2 -8739.296} C_VEL
LIN {X 0,Y 446.23,Z 591.432,A -85,B 0,C 180,E1 -8740.664,E2 -8740.664} C_VEL
LIN {X 0,Y 446.589,Z 582.767,A -85,B 0,C 180,E1 -8741.805,E2 -8741.805} C_VEL
LIN {X 0,Y 447.101,Z 573.652,A -85,B 0,C 180,E1 -8742.794,E2 -8742.794} C_VEL
LIN {X 0,Y 447.6,Z 563.03,A -85,B 0,C 180,E1 -8743.738,E2 -8743.738} C_VEL
LIN {X 0,Y 448.288,Z 551.887,A -85,B 0,C 180,E1 -8744.527,E2 -8744.527} C_VEL
LIN {X 0,Y 448.926,Z 539.56,A -85,B 0,C 180,E1 -8745.202,E2 -8745.202} C_VEL
LIN {X 0,Y 449.557,Z 526.655,A -85,B 0,C 180,E1 -8745.703,E2 -8745.703} C_VEL
LIN {X 0,Y 449.943,Z 512.986,A -85,B 0,C 180,E1 -8746.038,E2 -8746.038} C_VEL
LIN {X 0,Y 450.399,Z 435.658,A -85,B 0,C 180,E1 -8747.281,E2 -8747.281} C_VEL
LIN {X 0,Y 447.299,Z 407.056,A -85,B 0,C 180,E1 -8747.886,E2 -8747.886} C_VEL
LIN {X 0,Y 448.263,Z 381.806,A -85,B 0,C 180,E1 -8751.378,E2 -8751.378} C_VEL
LIN {X 0,Y 449.416,Z 357.314,A -85,B 0,C 180,E1 -8754.788,E2 -8754.788} C_VEL
LIN {X 0,Y 450.487,Z 335.221,A -85,B 0,C 180,E1 -8757.906,E2 -8757.906} C_VEL
LIN {X 0,Y 448.443,Z 324.493,A -85,B 0,C 180,E1 -8759.581,E2 -8759.581} C_VEL
LIN {X 0,Y 446.473,Z 315.994,A -85,B 0,C 180,E1 -8760.999,E2 -8760.999} C_VEL
LIN {X 0,Y 446.418,Z 315.877,A -85,B 0,C 180,E1 -8764.523,E2 -8764.523} C_VEL
LIN {X 0,Y 446.395,Z 315.879,A -85,B 0,C 180,E1 -8768.076,E2 -8768.076} C_VEL
LIN {X 0,Y 446.396,Z 315.877,A -85,B 0,C 180,E1 -8771.394,E2 -8771.394} C_VEL
LIN {X 0,Y 446.417,Z 315.854,A -85,B 0,C 180,E1 -8775.107,E2 -8775.107} C_VEL
LIN {X 0,Y 446.397,Z 315.878,A -85,B 0,C 180,E1 -8778.605,E2 -8778.605} C_VEL
LIN {X 0,Y 446.392,Z 315.851,A -85,B 0,C 180,E1 -8781.923,E2 -8781.923} C_VEL
LIN {X 0,Y 446.414,Z 315.863,A -85,B 0,C 180,E1 -8785.476,E2 -8785.476} C_VEL
LIN {X 0,Y 446.408,Z 315.875,A -85,B 0,C 180,E1 -8788.699,E2 -8788.699} C_VEL
LIN {X 0,Y 446.442,Z 315.864,A -85,B 0,C 180,E1 -8791.83,E2 -8791.83} C_VEL
LIN {X 0,Y 446.414,Z 315.874,A -85,B 0,C 180,E1 -8794.845,E2 -8794.845} C_VEL
LIN {X 0,Y 446.441,Z 315.859,A -85,B 0,C 180,E1 -8798.245,E2 -8798.245} C_VEL
LIN {X 0,Y 446.443,Z 315.868,A -85,B 0,C 180,E1 -8801.649,E2 -8801.649} C_VEL
LIN {X 0,Y 446.5,Z 315.863,A -85,B 0,C 180,E1 -8804.479,E2 -8804.479} C_VEL
LIN {X 0,Y 446.508,Z 315.862,A -85,B 0,C 180,E1 -8808.193,E2 -8808.193} C_VEL
LIN {X 0,Y 446.518,Z 315.861,A -85,B 0,C 180,E1 -8810.944,E2 -8810.944} C_VEL
LIN {X 0,Y 446.617,Z 315.845,A -85,B 0,C 180,E1 -8813.676,E2 -8813.676} C_VEL
LIN {X 0,Y 446.644,Z 315.848,A -85,B 0,C 180,E1 -8817.294,E2 -8817.294} C_VEL
LIN {X 0,Y 446.708,Z 315.831,A -85,B 0,C 180,E1 -8820,E2 -8820} C_VEL
LIN {X 0,Y 446.655,Z 315.841,A -85,B 0,C 180,E1 -8822.706,E2 -8822.706} C_VEL
LIN {X 0,Y 446.599,Z 315.847,A -85,B 0,C 180,E1 -8826.324,E2 -8826.324} C_VEL
LIN {X 0,Y 446.522,Z 315.855,A -85,B 0,C 180,E1 -8829.056,E2 -8829.056} C_VEL
LIN {X 0,Y 446.514,Z 315.859,A -85,B 0,C 180,E1 -8832.73,E2 -8832.73} C_VEL
LIN {X 0,Y 446.477,Z 315.865,A -85,B 0,C 180,E1 -8836.46,E2 -8836.46} C_VEL
LIN {X 0,Y 446.461,Z 315.872,A -85,B 0,C 180,E1 -8839.304,E2 -8839.304} C_VEL
LIN {X 0,Y 446.409,Z 315.874,A -85,B 0,C 180,E1 -8842.2,E2 -8842.2} C_VEL
LIN {X 0,Y 446.414,Z 315.877,A -85,B 0,C 180,E1 -8845.155,E2 -8845.155} C_VEL
LIN {X 0,Y 446.41,Z 315.855,A -85,B 0,C 180,E1 -8848.184,E2 -8848.184} C_VEL
LIN {X 0,Y 446.402,Z 315.86,A -85,B 0,C 180,E1 -8851.302,E2 -8851.302} C_VEL
LIN {X 0,Y 446.416,Z 315.874,A -85,B 0,C 180,E1 -8854.524,E2 -8854.524} C_VEL
LIN {X 0,Y 446.399,Z 315.862,A -85,B 0,C 180,E1 -8858.078,E2 -8858.078} C_VEL
LIN {X 0,Y 446.395,Z 315.873,A -85,B 0,C 180,E1 -8861.395,E2 -8861.395} C_VEL
LIN {X 0,Y 446.445,Z 315.872,A -85,B 0,C 180,E1 -8865.105,E2 -8865.105} C_VEL
LIN {X 0,Y 446.396,Z 315.873,A -85,B 0,C 180,E1 -8868.606,E2 -8868.606} C_VEL
LIN {X 0,Y 446.399,Z 315.869,A -85,B 0,C 180,E1 -8871.924,E2 -8871.924} C_VEL
LIN {X 0,Y 446.42,Z 315.879,A -85,B 0,C 180,E1 -8875.477,E2 -8875.477} C_VEL
LIN {X 0,Y 446.391,Z 315.877,A -85,B 0,C 180,E1 -8878.698,E2 -8878.698} C_VEL
LIN {X 0,Y 446.405,Z 315.858,A -85,B 0,C 180,E1 -8881.841,E2 -8881.841} C_VEL
LIN {X 0,Y 446.412,Z 315.877,A -85,B 0,C 180,E1 -8884.845,E2 -8884.845} C_VEL
LIN {X 0,Y 446.449,Z 315.86,A -85,B 0,C 180,E1 -8888.246,E2 -8888.246} C_VEL
LIN {X 0,Y 446.426,Z 315.834,A -85,B 0,C 180,E1 -8891.648,E2 -8891.648} C_VEL
LIN {X 0,Y 446.515,Z 316.095,A -85,B 0,C 180,E1 -8892.481,E2 -8892.481} C_VEL
LIN {X 0,Y 446.76,Z 317.173,A -85,B 0,C 180,E1 -8892.62,E2 -8892.62} C_VEL
LIN {X 0,Y 451.114,Z 328.721,A -85,B 0,C 180,E1 -8893.005,E2 -8893.005} C_VEL
LIN {X 0,Y 450.738,Z 397.348,A -85,B 0,C 180,E1 -8894.137,E2 -8894.137} C_VEL
LIN {X 0,Y 450.593,Z 410.385,A -85,B 0,C 180,E1 -8894.537,E2 -8894.537} C_VEL
LIN {X 0,Y 450.384,Z 422.363,A -85,B 0,C 180,E1 -8895.081,E2 -8895.081} C_VEL
LIN {X 0,Y 450.27,Z 425.89,A -85,B 0,C 180,E1 -8895.276,E2 -8895.276} C_VEL
LIN {X 0,Y 449.446,Z 431.286,A -85,B 0,C 180,E1 -8895.578,E2 -8895.578} C_VEL
LIN {X 0,Y 446.464,Z 439.878,A -85,B 0,C 180,E1 -8896.08,E2 -8896.08} C_VEL
LIN {X 0,Y 443.324,Z 448.083,A -85,B 0,C 180,E1 -8896.663,E2 -8896.663} C_VEL
LIN {X 0,Y 442.245,Z 452.805,A -85,B 0,C 180,E1 -8897.089,E2 -8897.089} C_VEL
LIN {X 0,Y 441.774,Z 461.418,A -85,B 0,C 180,E1 -8898.065,E2 -8898.065} C_VEL
LIN {X 0,Y 441.342,Z 469.79,A -85,B 0,C 180,E1 -8899.216,E2 -8899.216} C_VEL
LIN {X 0,Y 440.762,Z 477.921,A -85,B 0,C 180,E1 -8900.594,E2 -8900.594} C_VEL
LIN {X 0,Y 440.248,Z 485.038,A -85,B 0,C 180,E1 -8902.107,E2 -8902.107} C_VEL
LIN {X 0,Y 440.004,Z 490.422,A -85,B 0,C 180,E1 -8903.581,E2 -8903.581} C_VEL
LIN {X 0,Y 439.617,Z 494.318,A -85,B 0,C 180,E1 -8904.956,E2 -8904.956} C_VEL
LIN {X 0,Y 439.368,Z 497.188,A -85,B 0,C 180,E1 -8906.332,E2 -8906.332} C_VEL
LIN {X 0,Y 439.41,Z 498.543,A -85,B 0,C 180,E1 -8907.25,E2 -8907.25} C_VEL
LIN {X 0,Y 439.269,Z 499.529,A -85,B 0,C 180,E1 -8908.166,E2 -8908.166} C_VEL
LIN {X 0,Y 439.349,Z 500.113,A -85,B 0,C 180,E1 -8909.083,E2 -8909.083} C_VEL
LIN {X 0,Y 439.332,Z 500.344,A -85,B 0,C 180,E1 -8910,E2 -8910} C_VEL
LIN {X 0,Y 439.349,Z 500.161,A -85,B 0,C 180,E1 -8910.917,E2 -8910.917} C_VEL
LIN {X 0,Y 439.269,Z 499.606,A -85,B 0,C 180,E1 -8911.834,E2 -8911.834} C_VEL
LIN {X 0,Y 439.408,Z 498.652,A -85,B 0,C 180,E1 -8912.75,E2 -8912.75} C_VEL
LIN {X 0,Y 439.362,Z 497.346,A -85,B 0,C 180,E1 -8913.668,E2 -8913.668} C_VEL
LIN {X 0,Y 439.611,Z 494.534,A -85,B 0,C 180,E1 -8915.044,E2 -8915.044} C_VEL
LIN {X 0,Y 439.987,Z 490.713,A -85,B 0,C 180,E1 -8916.42,E2 -8916.42} C_VEL
LIN {X 0,Y 440.198,Z 485.638,A -85,B 0,C 180,E1 -8917.846,E2 -8917.846} C_VEL
LIN {X 0,Y 440.758,Z 478.409,A -85,B 0,C 180,E1 -8919.406,E2 -8919.406} C_VEL
LIN {X 0,Y 441.333,Z 470.384,A -85,B 0,C 180,E1 -8920.784,E2 -8920.784} C_VEL
LIN {X 0,Y 441.794,Z 462.166,A -85,B 0,C 180,E1 -8921.935,E2 -8921.935} C_VEL
LIN {X 0,Y 442.297,Z 453.141,A -85,B 0,C 180,E1 -8922.97,E2 -8922.97} C_VEL
LIN {X 0,Y 442.923,Z 442.645,A -85,B 0,C 180,E1 -8923.939,E2 -8923.939} C_VEL
LIN {X 0,Y 443.318,Z 431.151,A -85,B 0,C 180,E1 -8924.788,E2 -8924.788} C_VEL
LIN {X 0,Y 443.672,Z 419.909,A -85,B 0,C 180,E1 -8925.427,E2 -8925.427} C_VEL
LIN {X 0,Y 443.872,Z 406.736,A -85,B 0,C 180,E1 -8925.968,E2 -8925.968} C_VEL
LIN {X 0,Y 443.902,Z 393.008,A -85,B 0,C 180,E1 -8926.321,E2 -8926.321} C_VEL
LIN {X 0,Y 444.321,Z 330.1,A -85,B 0,C 180,E1 -8927.353,E2 -8927.353} C_VEL
LIN {X 0,Y 439.608,Z 317.698,A -85,B 0,C 180,E1 -8927.79,E2 -8927.79} C_VEL
LIN {X 0,Y 439.423,Z 316.841,A -85,B 0,C 180,E1 -8927.961,E2 -8927.961} C_VEL
LIN {X 0,Y 439.376,Z 316.758,A -85,B 0,C 180,E1 -8930.603,E2 -8930.603} C_VEL
LIN {X 0,Y 439.365,Z 316.751,A -85,B 0,C 180,E1 -8933.571,E2 -8933.571} C_VEL
LIN {X 0,Y 439.354,Z 316.736,A -85,B 0,C 180,E1 -8936.608,E2 -8936.608} C_VEL
LIN {X 0,Y 439.367,Z 316.751,A -85,B 0,C 180,E1 -8939.726,E2 -8939.726} C_VEL
LIN {X 0,Y 439.34,Z 316.754,A -85,B 0,C 180,E1 -8942.948,E2 -8942.948} C_VEL
LIN {X 0,Y 439.366,Z 316.754,A -85,B 0,C 180,E1 -8946.287,E2 -8946.287} C_VEL
LIN {X 0,Y 439.356,Z 316.754,A -85,B 0,C 180,E1 -8949.779,E2 -8949.779} C_VEL
LIN {X 0,Y 439.325,Z 316.748,A -85,B 0,C 180,E1 -8952.619,E2 -8952.619} C_VEL
LIN {X 0,Y 439.392,Z 316.749,A -85,B 0,C 180,E1 -8955.269,E2 -8955.269} C_VEL
LIN {X 0,Y 439.348,Z 316.747,A -85,B 0,C 180,E1 -8959.015,E2 -8959.015} C_VEL
LIN {X 0,Y 439.336,Z 316.747,A -85,B 0,C 180,E1 -8962.563,E2 -8962.563} C_VEL
LIN {X 0,Y 439.389,Z 316.754,A -85,B 0,C 180,E1 -8964.843,E2 -8964.843} C_VEL
LIN {X 0,Y 439.363,Z 316.748,A -85,B 0,C 180,E1 -8968.139,E2 -8968.139} C_VEL
LIN {X 0,Y 439.38,Z 316.73,A -85,B 0,C 180,E1 -8971.609,E2 -8971.609} C_VEL
LIN {X 0,Y 439.359,Z 316.753,A -85,B 0,C 180,E1 -8974.412,E2 -8974.412} C_VEL
LIN {X 0,Y 439.346,Z 316.752,A -85,B 0,C 180,E1 -8977.423,E2 -8977.423} C_VEL
LIN {X 0,Y 439.434,Z 316.748,A -85,B 0,C 180,E1 -8980.663,E2 -8980.663} C_VEL
LIN {X 0,Y 439.446,Z 316.744,A -85,B 0,C 180,E1 -8984.224,E2 -8984.224} C_VEL
LIN {X 0,Y 439.474,Z 316.739,A -85,B 0,C 180,E1 -8988.001,E2 -8988.001} C_VEL
LIN {X 0,Y 439.472,Z 316.733,A -85,B 0,C 180,E1 -8991.725,E2 -8991.725} C_VEL
LIN {X 0,Y 439.583,Z 316.73,A -85,B 0,C 180,E1 -8994.495,E2 -8994.495} C_VEL
LIN {X 0,Y 439.621,Z 316.719,A -85,B 0,C 180,E1 -8998.168,E2 -8998.168} C_VEL
LIN {X 0,Y 439.576,Z 316.725,A -85,B 0,C 180,E1 -9000.916,E2 -9000.916} C_VEL
LIN {X 0,Y 439.595,Z 316.725,A -85,B 0,C 180,E1 -9002.749,E2 -9002.749} C_VEL
LIN {X 0,Y 439.587,Z 316.72,A -85,B 0,C 180,E1 -9006.426,E2 -9006.426} C_VEL
LIN {X 0,Y 439.474,Z 316.738,A -85,B 0,C 180,E1 -9009.202,E2 -9009.202} C_VEL
LIN {X 0,Y 439.458,Z 316.733,A -85,B 0,C 180,E1 -9012.938,E2 -9012.938} C_VEL
LIN {X 0,Y 439.438,Z 316.748,A -85,B 0,C 180,E1 -9016.348,E2 -9016.348} C_VEL
LIN {X 0,Y 439.395,Z 316.74,A -85,B 0,C 180,E1 -9019.627,E2 -9019.627} C_VEL
LIN {X 0,Y 439.356,Z 316.754,A -85,B 0,C 180,E1 -9022.576,E2 -9022.576} C_VEL
LIN {X 0,Y 439.359,Z 316.754,A -85,B 0,C 180,E1 -9025.588,E2 -9025.588} C_VEL
LIN {X 0,Y 439.39,Z 316.742,A -85,B 0,C 180,E1 -9028.675,E2 -9028.675} C_VEL
LIN {X 0,Y 439.361,Z 316.76,A -85,B 0,C 180,E1 -9032.03,E2 -9032.03} C_VEL
LIN {X 0,Y 439.381,Z 316.745,A -85,B 0,C 180,E1 -9035.339,E2 -9035.339} C_VEL
LIN {X 0,Y 439.349,Z 316.751,A -85,B 0,C 180,E1 -9038.599,E2 -9038.599} C_VEL
LIN {X 0,Y 439.347,Z 316.757,A -85,B 0,C 180,E1 -9042.21,E2 -9042.21} C_VEL
LIN {X 0,Y 439.368,Z 316.732,A -85,B 0,C 180,E1 -9045.267,E2 -9045.267} C_VEL
LIN {X 0,Y 439.359,Z 316.752,A -85,B 0,C 180,E1 -9048.748,E2 -9048.748} C_VEL
LIN {X 0,Y 439.353,Z 316.752,A -85,B 0,C 180,E1 -9051.612,E2 -9051.612} C_VEL
LIN {X 0,Y 439.388,Z 316.747,A -85,B 0,C 180,E1 -9054.844,E2 -9054.844} C_VEL
LIN {X 0,Y 439.368,Z 316.756,A -85,B 0,C 180,E1 -9058.14,E2 -9058.14} C_VEL
LIN {X 0,Y 439.453,Z 317.061,A -85,B 0,C 180,E1 -9058.768,E2 -9058.768} C_VEL
LIN {X 0,Y 443.062,Z 333.058,A -85,B 0,C 180,E1 -9061.401,E2 -9061.401} C_VEL
LIN {X 0,Y 443.598,Z 336.273,A -85,B 0,C 180,E1 -9061.905,E2 -9061.905} C_VEL
LIN {X 0,Y 442.523,Z 357.656,A -85,B 0,C 180,E1 -9064.975,E2 -9064.975} C_VEL
LIN {X 0,Y 441.433,Z 379.193,A -85,B 0,C 180,E1 -9068.029,E2 -9068.029} C_VEL
LIN {X 0,Y 440.423,Z 402.836,A -85,B 0,C 180,E1 -9071.389,E2 -9071.389} C_VEL
LIN {X 0,Y 440.311,Z 405.918,A -85,B 0,C 180,E1 -9071.807,E2 -9071.807} C_VEL
LIN {X 0,Y 443.701,Z 438.301,A -85,B 0,C 180,E1 -9072.506,E2 -9072.506} C_VEL
LIN {X 0,Y 442.967,Z 516.501,A -85,B 0,C 180,E1 -9073.792,E2 -9073.792} C_VEL
LIN {X 0,Y 442.459,Z 529.814,A -85,B 0,C 180,E1 -9074.187,E2 -9074.187} C_VEL
LIN {X 0,Y 441.749,Z 543.17,A -85,B 0,C 180,E1 -9074.781,E2 -9074.781} C_VEL
LIN {X 0,Y 441.147,Z 554.426,A -85,B 0,C 180,E1 -9075.469,E2 -9075.469} C_VEL
LIN {X 0,Y 440.509,Z 564.974,A -85,B 0,C 180,E1 -9076.284,E2 -9076.284} C_VEL
LIN {X 0,Y 440.041,Z 575.681,A -85,B 0,C 180,E1 -9077.314,E2 -9077.314} C_VEL
LIN {X 0,Y 439.38,Z 585.44,A -85,B 0,C 180,E1 -9078.467,E2 -9078.467} C_VEL
LIN {X 0,Y 439.061,Z 593.492,A -85,B 0,C 180,E1 -9079.626,E2 -9079.626} C_VEL
LIN {X 0,Y 438.788,Z 601.38,A -85,B 0,C 180,E1 -9081.016,E2 -9081.016} C_VEL
LIN {X 0,Y 438.717,Z 606.805,A -85,B 0,C 180,E1 -9082.174,E2 -9082.174} C_VEL
LIN {X 0,Y 438.685,Z 612.075,A -85,B 0,C 180,E1 -9083.561,E2 -9083.561} C_VEL
LIN {X 0,Y 438.757,Z 616.183,A -85,B 0,C 180,E1 -9084.946,E2 -9084.946} C_VEL
LIN {X 0,Y 438.839,Z 619.222,A -85,B 0,C 180,E1 -9086.327,E2 -9086.327} C_VEL
LIN {X 0,Y 438.825,Z 620.664,A -85,B 0,C 180,E1 -9087.246,E2 -9087.246} C_VEL
LIN {X 0,Y 439.032,Z 622.35,A -85,B 0,C 180,E1 -9089.083,E2 -9089.083} C_VEL
LIN {X 0,Y 439.032,Z 622.573,A -85,B 0,C 180,E1 -9090,E2 -9090} C_VEL
LIN {X 0,Y 439.032,Z 622.349,A -85,B 0,C 180,E1 -9090.917,E2 -9090.917} C_VEL
LIN {X 0,Y 438.825,Z 620.665,A -85,B 0,C 180,E1 -9092.754,E2 -9092.754} C_VEL
LIN {X 0,Y 438.839,Z 619.223,A -85,B 0,C 180,E1 -9093.673,E2 -9093.673} C_VEL
LIN {X 0,Y 438.759,Z 616.18,A -85,B 0,C 180,E1 -9095.054,E2 -9095.054} C_VEL
LIN {X 0,Y 438.727,Z 611.177,A -85,B 0,C 180,E1 -9096.693,E2 -9096.693} C_VEL
LIN {X 0,Y 438.757,Z 604.729,A -85,B 0,C 180,E1 -9098.289,E2 -9098.289} C_VEL
LIN {X 0,Y 438.891,Z 597.639,A -85,B 0,C 180,E1 -9099.679,E2 -9099.679} C_VEL
LIN {X 0,Y 439.255,Z 588.808,A -85,B 0,C 180,E1 -9101.069,E2 -9101.069} C_VEL
LIN {X 0,Y 439.791,Z 579.798,A -85,B 0,C 180,E1 -9102.224,E2 -9102.224} C_VEL
LIN {X 0,Y 440.314,Z 569.204,A -85,B 0,C 180,E1 -9103.335,E2 -9103.335} C_VEL
LIN {X 0,Y 440.885,Z 557.573,A -85,B 0,C 180,E1 -9104.305,E2 -9104.305} C_VEL
LIN {X 0,Y 441.7,Z 545.152,A -85,B 0,C 180,E1 -9105.102,E2 -9105.102} C_VEL
LIN {X 0,Y 442.291,Z 533.406,A -85,B 0,C 180,E1 -9105.672,E2 -9105.672} C_VEL
LIN {X 0,Y 442.843,Z 520.936,A -85,B 0,C 180,E1 -9106.095,E2 -9106.095} C_VEL
LIN {X 0,Y 443.128,Z 505.06,A -85,B 0,C 180,E1 -9106.41,E2 -9106.41} C_VEL
LIN {X 0,Y 443.565,Z 436.353,A -85,B 0,C 180,E1 -9107.527,E2 -9107.527} C_VEL
LIN {X 0,Y 440.307,Z 406.147,A -85,B 0,C 180,E1 -9108.173,E2 -9108.173} C_VEL
LIN {X 0,Y 441.276,Z 382.558,A -85,B 0,C 180,E1 -9111.488,E2 -9111.488} C_VEL
LIN {X 0,Y 442.505,Z 357.646,A -85,B 0,C 180,E1 -9115.02,E2 -9115.02} C_VEL
LIN {X 0,Y 443.592,Z 337.804,A -85,B 0,C 180,E1 -9117.863,E2 -9117.863} C_VEL
LIN {X 0,Y 443.003,Z 333.017,A -85,B 0,C 180,E1 -9118.602,E2 -9118.602} C_VEL
LIN {X 0,Y 439.714,Z 318.161,A -85,B 0,C 180,E1 -9121.027,E2 -9121.027} C_VEL
LIN {X 0,Y 439.388,Z 316.818,A -85,B 0,C 180,E1 -9121.321,E2 -9121.321} C_VEL
LIN {X 0,Y 439.356,Z 316.76,A -85,B 0,C 180,E1 -9124.046,E2 -9124.046} C_VEL
LIN {X 0,Y 439.335,Z 316.759,A -85,B 0,C 180,E1 -9126.884,E2 -9126.884} C_VEL
LIN {X 0,Y 439.342,Z 316.747,A -85,B 0,C 180,E1 -9129.84,E2 -9129.84} C_VEL
LIN {X 0,Y 439.329,Z 316.758,A -85,B 0,C 180,E1 -9132.619,E2 -9132.619} C_VEL
LIN {X 0,Y 439.371,Z 316.731,A -85,B 0,C 180,E1 -9135.267,E2 -9135.267} C_VEL
LIN {X 0,Y 439.359,Z 316.754,A -85,B 0,C 180,E1 -9138.746,E2 -9138.746} C_VEL
LIN {X 0,Y 439.35,Z 316.732,A -85,B 0,C 180,E1 -9141.61,E2 -9141.61} C_VEL
LIN {X 0,Y 439.386,Z 316.735,A -85,B 0,C 180,E1 -9144.843,E2 -9144.843} C_VEL
LIN {X 0,Y 439.364,Z 316.757,A -85,B 0,C 180,E1 -9148.139,E2 -9148.139} C_VEL
LIN {X 0,Y 439.397,Z 316.74,A -85,B 0,C 180,E1 -9151.605,E2 -9151.605} C_VEL
LIN {X 0,Y 439.359,Z 316.755,A -85,B 0,C 180,E1 -9154.412,E2 -9154.412} C_VEL
LIN {X 0,Y 439.356,Z 316.753,A -85,B 0,C 180,E1 -9157.424,E2 -9157.424} C_VEL
LIN {X 0,Y 439.434,Z 316.735,A -85,B 0,C 180,E1 -9160.663,E2 -9160.663} C_VEL
LIN {X 0,Y 439.454,Z 316.743,A -85,B 0,C 180,E1 -9164.224,E2 -9164.224} C_VEL
LIN {X 0,Y 439.475,Z 316.739,A -85,B 0,C 180,E1 -9168.001,E2 -9168.001} C_VEL
LIN {X 0,Y 439.494,Z 316.739,A -85,B 0,C 180,E1 -9171.725,E2 -9171.725} C_VEL
LIN {X 0,Y 439.6,Z 316.717,A -85,B 0,C 180,E1 -9174.496,E2 -9174.496} C_VEL
LIN {X 0,Y 439.617,Z 316.721,A -85,B 0,C 180,E1 -9178.168,E2 -9178.168} C_VEL
LIN {X 0,Y 439.659,Z 316.709,A -85,B 0,C 180,E1 -9180,E2 -9180} C_VEL
LIN {X 0,Y 439.607,Z 316.719,A -85,B 0,C 180,E1 -9182.749,E2 -9182.749} C_VEL
LIN {X 0,Y 439.551,Z 316.724,A -85,B 0,C 180,E1 -9186.426,E2 -9186.426} C_VEL
LIN {X 0,Y 439.486,Z 316.733,A -85,B 0,C 180,E1 -9189.202,E2 -9189.202} C_VEL
LIN {X 0,Y 439.458,Z 316.739,A -85,B 0,C 180,E1 -9192.938,E2 -9192.938} C_VEL
LIN {X 0,Y 439.437,Z 316.742,A -85,B 0,C 180,E1 -9196.347,E2 -9196.347} C_VEL
LIN {X 0,Y 439.394,Z 316.748,A -85,B 0,C 180,E1 -9199.627,E2 -9199.627} C_VEL
LIN {X 0,Y 439.355,Z 316.751,A -85,B 0,C 180,E1 -9202.576,E2 -9202.576} C_VEL
LIN {X 0,Y 439.36,Z 316.754,A -85,B 0,C 180,E1 -9205.588,E2 -9205.588} C_VEL
LIN {X 0,Y 439.374,Z 316.73,A -85,B 0,C 180,E1 -9208.677,E2 -9208.677} C_VEL
LIN {X 0,Y 439.36,Z 316.749,A -85,B 0,C 180,E1 -9212.03,E2 -9212.03} C_VEL
LIN {X 0,Y 439.385,Z 316.756,A -85,B 0,C 180,E1 -9215.34,E2 -9215.34} C_VEL
LIN {X 0,Y 439.352,Z 316.738,A -85,B 0,C 180,E1 -9218.598,E2 -9218.598} C_VEL
LIN {X 0,Y 439.344,Z 316.755,A -85,B 0,C 180,E1 -9222.211,E2 -9222.211} C_VEL
LIN {X 0,Y 439.393,Z 316.747,A -85,B 0,C 180,E1 -9225.271,E2 -9225.271} C_VEL
LIN {X 0,Y 439.35,Z 316.754,A -85,B 0,C 180,E1 -9229.017,E2 -9229.017} C_VEL
LIN {X 0,Y 439.336,Z 316.747,A -85,B 0,C 180,E1 -9232.564,E2 -9232.564} C_VEL
LIN {X 0,Y 439.392,Z 316.75,A -85,B 0,C 180,E1 -9234.844,E2 -9234.844} C_VEL
LIN {X 0,Y 439.351,Z 316.753,A -85,B 0,C 180,E1 -9238.138,E2 -9238.138} C_VEL
LIN {X 0,Y 439.379,Z 316.739,A -85,B 0,C 180,E1 -9241.324,E2 -9241.324} C_VEL
LIN {X 0,Y 439.353,Z 316.754,A -85,B 0,C 180,E1 -9244.412,E2 -9244.412} C_VEL
LIN {X 0,Y 439.362,Z 316.742,A -85,B 0,C 180,E1 -9247.425,E2 -9247.425} C_VEL
LIN {X 0,Y 439.442,Z 316.729,A -85,B 0,C 180,E1 -9250.664,E2 -9250.664} C_VEL
LIN {X 0,Y 439.447,Z 316.893,A -85,B 0,C 180,E1 -9252.16,E2 -9252.16} C_VEL
LIN {X 0,Y 439.666,Z 317.868,A -85,B 0,C 180,E1 -9252.32,E2 -9252.32} C_VEL
LIN {X 0,Y 444.414,Z 330.365,A -85,B 0,C 180,E1 -9252.751,E2 -9252.751} C_VEL
LIN {X 0,Y 443.969,Z 397.14,A -85,B 0,C 180,E1 -9253.859,E2 -9253.859} C_VEL
LIN {X 0,Y 443.858,Z 409.864,A -85,B 0,C 180,E1 -9254.238,E2 -9254.238} C_VEL
LIN {X 0,Y 443.589,Z 422.237,A -85,B 0,C 180,E1 -9254.788,E2 -9254.788} C_VEL
LIN {X 0,Y 443.239,Z 434.595,A -85,B 0,C 180,E1 -9255.537,E2 -9255.537} C_VEL
LIN {X 0,Y 442.618,Z 446.18,A -85,B 0,C 180,E1 -9256.456,E2 -9256.456} C_VEL
LIN {X 0,Y 442.245,Z 452.805,A -85,B 0,C 180,E1 -9257.089,E2 -9257.089} C_VEL
LIN {X 0,Y 441.151,Z 457.469,A -85,B 0,C 180,E1 -9257.545,E2 -9257.545} C_VEL
LIN {X 0,Y 437.915,Z 464.803,A -85,B 0,C 180,E1 -9258.314,E2 -9258.314} C_VEL
LIN {X 0,Y 434.856,Z 471.529,A -85,B 0,C 180,E1 -9259.175,E2 -9259.175} C_VEL
LIN {X 0,Y 434.044,Z 475.232,A -85,B 0,C 180,E1 -9259.77,E2 -9259.77} C_VEL
LIN {X 0,Y 433.559,Z 482.567,A -85,B 0,C 180,E1 -9261.189,E2 -9261.189} C_VEL
LIN {X 0,Y 433.205,Z 488.184,A -85,B 0,C 180,E1 -9262.543,E2 -9262.543} C_VEL
LIN {X 0,Y 432.805,Z 492.806,A -85,B 0,C 180,E1 -9263.941,E2 -9263.941} C_VEL
LIN {X 0,Y 432.501,Z 496.342,A -85,B 0,C 180,E1 -9265.34,E2 -9265.34} C_VEL
LIN {X 0,Y 432.351,Z 498.167,A -85,B 0,C 180,E1 -9266.272,E2 -9266.272} C_VEL
LIN {X 0,Y 432.391,Z 499.521,A -85,B 0,C 180,E1 -9267.205,E2 -9267.205} C_VEL
LIN {X 0,Y 432.247,Z 500.507,A -85,B 0,C 180,E1 -9268.137,E2 -9268.137} C_VEL
LIN {X 0,Y 432.326,Z 501.091,A -85,B 0,C 180,E1 -9269.069,E2 -9269.069} C_VEL
LIN {X 0,Y 432.31,Z 501.322,A -85,B 0,C 180,E1 -9270,E2 -9270} C_VEL
LIN {X 0,Y 432.326,Z 501.138,A -85,B 0,C 180,E1 -9270.931,E2 -9270.931} C_VEL
LIN {X 0,Y 432.247,Z 500.584,A -85,B 0,C 180,E1 -9271.863,E2 -9271.863} C_VEL
LIN {X 0,Y 432.389,Z 499.629,A -85,B 0,C 180,E1 -9272.795,E2 -9272.795} C_VEL
LIN {X 0,Y 432.344,Z 498.324,A -85,B 0,C 180,E1 -9273.728,E2 -9273.728} C_VEL
LIN {X 0,Y 432.608,Z 495.512,A -85,B 0,C 180,E1 -9275.126,E2 -9275.126} C_VEL
LIN {X 0,Y 433.005,Z 491.69,A -85,B 0,C 180,E1 -9276.524,E2 -9276.524} C_VEL
LIN {X 0,Y 433.236,Z 486.615,A -85,B 0,C 180,E1 -9277.972,E2 -9277.972} C_VEL
LIN {X 0,Y 433.827,Z 479.385,A -85,B 0,C 180,E1 -9279.558,E2 -9279.558} C_VEL
LIN {X 0,Y 434.432,Z 471.359,A -85,B 0,C 180,E1 -9280.958,E2 -9280.958} C_VEL
LIN {X 0,Y 434.918,Z 463.141,A -85,B 0,C 180,E1 -9282.126,E2 -9282.126} C_VEL
LIN {X 0,Y 435.435,Z 454.117,A -85,B 0,C 180,E1 -9283.178,E2 -9283.178} C_VEL
LIN {X 0,Y 436.105,Z 443.617,A -85,B 0,C 180,E1 -9284.161,E2 -9284.161} C_VEL
LIN {X 0,Y 436.529,Z 431.968,A -85,B 0,C 180,E1 -9285.034,E2 -9285.034} C_VEL
LIN {X 0,Y 436.916,Z 420.544,A -85,B 0,C 180,E1 -9285.69,E2 -9285.69} C_VEL
LIN {X 0,Y 437.106,Z 407.702,A -85,B 0,C 180,E1 -9286.222,E2 -9286.222} C_VEL
LIN {X 0,Y 437.141,Z 393.966,A -85,B 0,C 180,E1 -9286.581,E2 -9286.581} C_VEL
LIN {X 0,Y 437.562,Z 331.587,A -85,B 0,C 180,E1 -9287.621,E2 -9287.621} C_VEL
LIN {X 0,Y 432.583,Z 318.692,A -85,B 0,C 180,E1 -9288.082,E2 -9288.082} C_VEL
LIN {X 0,Y 432.368,Z 317.721,A -85,B 0,C 180,E1 -9288.265,E2 -9288.265} C_VEL
LIN {X 0,Y 432.343,Z 317.628,A -85,B 0,C 180,E1 -9290.954,E2 -9290.954} C_VEL
LIN {X 0,Y 432.347,Z 317.63,A -85,B 0,C 180,E1 -9294.452,E2 -9294.452} C_VEL
LIN {X 0,Y 432.313,Z 317.611,A -85,B 0,C 180,E1 -9298.128,E2 -9298.128} C_VEL
LIN {X 0,Y 432.3,Z 317.632,A -85,B 0,C 180,E1 -9301.347,E2 -9301.347} C_VEL
LIN {X 0,Y 432.322,Z 317.636,A -85,B 0,C 180,E1 -9304.678,E2 -9304.678} C_VEL
LIN {X 0,Y 432.322,Z 317.622,A -85,B 0,C 180,E1 -9308.151,E2 -9308.151} C_VEL
LIN {X 0,Y 432.299,Z 317.629,A -85,B 0,C 180,E1 -9311.8,E2 -9311.8} C_VEL
LIN {X 0,Y 432.33,Z 317.619,A -85,B 0,C 180,E1 -9314.347,E2 -9314.347} C_VEL
LIN {X 0,Y 432.296,Z 317.636,A -85,B 0,C 180,E1 -9317.018,E2 -9317.018} C_VEL
LIN {X 0,Y 432.284,Z 317.624,A -85,B 0,C 180,E1 -9319.827,E2 -9319.827} C_VEL
LIN {X 0,Y 432.297,Z 317.632,A -85,B 0,C 180,E1 -9323.021,E2 -9323.021} C_VEL
LIN {X 0,Y 432.327,Z 317.631,A -85,B 0,C 180,E1 -9326.001,E2 -9326.001} C_VEL
LIN {X 0,Y 432.334,Z 317.606,A -85,B 0,C 180,E1 -9329.491,E2 -9329.491} C_VEL
LIN {X 0,Y 432.313,Z 317.61,A -85,B 0,C 180,E1 -9331.872,E2 -9331.872} C_VEL
LIN {X 0,Y 432.316,Z 317.632,A -85,B 0,C 180,E1 -9334.996,E2 -9334.996} C_VEL
LIN {X 0,Y 432.345,Z 317.627,A -85,B 0,C 180,E1 -9338.045,E2 -9338.045} C_VEL
LIN {X 0,Y 432.375,Z 317.624,A -85,B 0,C 180,E1 -9341.029,E2 -9341.029} C_VEL
LIN {X 0,Y 432.417,Z 317.618,A -85,B 0,C 180,E1 -9343.961,E2 -9343.961} C_VEL
LIN {X 0,Y 432.451,Z 317.613,A -85,B 0,C 180,E1 -9347.803,E2 -9347.803} C_VEL
LIN {X 0,Y 432.439,Z 317.608,A -85,B 0,C 180,E1 -9351.589,E2 -9351.589} C_VEL
LIN {X 0,Y 432.538,Z 317.606,A -85,B 0,C 180,E1 -9354.405,E2 -9354.405} C_VEL
LIN {X 0,Y 432.591,Z 317.595,A -85,B 0,C 180,E1 -9358.138,E2 -9358.138} C_VEL
LIN {X 0,Y 432.537,Z 317.602,A -85,B 0,C 180,E1 -9360.931,E2 -9360.931} C_VEL
LIN {X 0,Y 432.549,Z 317.603,A -85,B 0,C 180,E1 -9362.794,E2 -9362.794} C_VEL
LIN {X 0,Y 432.576,Z 317.591,A -85,B 0,C 180,E1 -9365.594,E2 -9365.594} C_VEL
LIN {X 0,Y 432.453,Z 317.618,A -85,B 0,C 180,E1 -9368.41,E2 -9368.41} C_VEL
LIN {X 0,Y 432.446,Z 317.611,A -85,B 0,C 180,E1 -9372.197,E2 -9372.197} C_VEL
LIN {X 0,Y 432.422,Z 317.621,A -85,B 0,C 180,E1 -9376.039,E2 -9376.039} C_VEL
LIN {X 0,Y 432.38,Z 317.613,A -85,B 0,C 180,E1 -9379.485,E2 -9379.485} C_VEL
LIN {X 0,Y 432.305,Z 317.629,A -85,B 0,C 180,E1 -9382.965,E2 -9382.965} C_VEL
LIN {X 0,Y 432.314,Z 317.635,A -85,B 0,C 180,E1 -9386.036,E2 -9386.036} C_VEL
LIN {X 0,Y 432.325,Z 317.621,A -85,B 0,C 180,E1 -9389.189,E2 -9389.189} C_VEL
LIN {X 0,Y 432.316,Z 317.632,A -85,B 0,C 180,E1 -9392.444,E2 -9392.444} C_VEL
LIN {X 0,Y 432.327,Z 317.627,A -85,B 0,C 180,E1 -9395.819,E2 -9395.819} C_VEL
LIN {X 0,Y 432.295,Z 317.628,A -85,B 0,C 180,E1 -9399.349,E2 -9399.349} C_VEL
LIN {X 0,Y 432.3,Z 317.637,A -85,B 0,C 180,E1 -9401.801,E2 -9401.801} C_VEL
LIN {X 0,Y 432.328,Z 317.61,A -85,B 0,C 180,E1 -9404.348,E2 -9404.348} C_VEL
LIN {X 0,Y 432.297,Z 317.632,A -85,B 0,C 180,E1 -9407.019,E2 -9407.019} C_VEL
LIN {X 0,Y 432.285,Z 317.627,A -85,B 0,C 180,E1 -9409.829,E2 -9409.829} C_VEL
LIN {X 0,Y 432.293,Z 317.635,A -85,B 0,C 180,E1 -9413.021,E2 -9413.021} C_VEL
LIN {X 0,Y 432.33,Z 317.633,A -85,B 0,C 180,E1 -9416.003,E2 -9416.003} C_VEL
LIN {X 0,Y 432.358,Z 317.824,A -85,B 0,C 180,E1 -9418.453,E2 -9418.453} C_VEL
LIN {X 0,Y 435.942,Z 333.38,A -85,B 0,C 180,E1 -9421.077,E2 -9421.077} C_VEL
LIN {X 0,Y 436.712,Z 338.701,A -85,B 0,C 180,E1 -9421.92,E2 -9421.92} C_VEL
LIN {X 0,Y 435.41,Z 361.1,A -85,B 0,C 180,E1 -9425.187,E2 -9425.187} C_VEL
LIN {X 0,Y 434.334,Z 381.637,A -85,B 0,C 180,E1 -9428.151,E2 -9428.151} C_VEL
LIN {X 0,Y 433.335,Z 404.944,A -85,B 0,C 180,E1 -9431.506,E2 -9431.506} C_VEL
LIN {X 0,Y 436.896,Z 438.811,A -85,B 0,C 180,E1 -9432.25,E2 -9432.25} C_VEL
LIN {X 0,Y 436.125,Z 515.521,A -85,B 0,C 180,E1 -9433.53,E2 -9433.53} C_VEL
LIN {X 0,Y 435.644,Z 528.836,A -85,B 0,C 180,E1 -9433.933,E2 -9433.933} C_VEL
LIN {X 0,Y 434.911,Z 542.188,A -85,B 0,C 180,E1 -9434.536,E2 -9434.536} C_VEL
LIN {X 0,Y 434.26,Z 553.439,A -85,B 0,C 180,E1 -9435.233,E2 -9435.233} C_VEL
LIN {X 0,Y 433.54,Z 563.979,A -85,B 0,C 180,E1 -9436.059,E2 -9436.059} C_VEL
LIN {X 0,Y 433.001,Z 573.939,A -85,B 0,C 180,E1 -9437.024,E2 -9437.024} C_VEL
LIN {X 0,Y 432.47,Z 582.629,A -85,B 0,C 180,E1 -9438.042,E2 -9438.042} C_VEL
LIN {X 0,Y 431.998,Z 592.495,A -85,B 0,C 180,E1 -9439.454,E2 -9439.454} C_VEL
LIN {X 0,Y 431.722,Z 600.385,A -85,B 0,C 180,E1 -9440.868,E2 -9440.868} C_VEL
LIN {X 0,Y 431.65,Z 605.813,A -85,B 0,C 180,E1 -9442.045,E2 -9442.045} C_VEL
LIN {X 0,Y 431.611,Z 611.085,A -85,B 0,C 180,E1 -9443.455,E2 -9443.455} C_VEL
LIN {X 0,Y 431.689,Z 615.196,A -85,B 0,C 180,E1 -9444.863,E2 -9444.863} C_VEL
LIN {X 0,Y 431.796,Z 618.241,A -85,B 0,C 180,E1 -9446.267,E2 -9446.267} C_VEL
LIN {X 0,Y 431.779,Z 619.682,A -85,B 0,C 180,E1 -9447.201,E2 -9447.201} C_VEL
LIN {X 0,Y 432.004,Z 621.372,A -85,B 0,C 180,E1 -9449.068,E2 -9449.068} C_VEL
LIN {X 0,Y 432.009,Z 621.596,A -85,B 0,C 180,E1 -9450,E2 -9450} C_VEL
LIN {X 0,Y 432.004,Z 621.371,A -85,B 0,C 180,E1 -9450.932,E2 -9450.932} C_VEL
LIN {X 0,Y 431.779,Z 619.683,A -85,B 0,C 180,E1 -9452.799,E2 -9452.799} C_VEL
LIN {X 0,Y 431.796,Z 618.24,A -85,B 0,C 180,E1 -9453.733,E2 -9453.733} C_VEL
LIN {X 0,Y 431.692,Z 615.192,A -85,B 0,C 180,E1 -9455.137,E2 -9455.137} C_VEL
LIN {X 0,Y 431.664,Z 610.526,A -85,B 0,C 180,E1 -9456.708,E2 -9456.708} C_VEL
LIN {X 0,Y 431.678,Z 603.732,A -85,B 0,C 180,E1 -9458.425,E2 -9458.425} C_VEL
LIN {X 0,Y 431.817,Z 596.638,A -85,B 0,C 180,E1 -9459.839,E2 -9459.839} C_VEL
LIN {X 0,Y 432.23,Z 587.809,A -85,B 0,C 180,E1 -9461.251,E2 -9461.251} C_VEL
LIN {X 0,Y 432.806,Z 578.866,A -85,B 0,C 180,E1 -9462.417,E2 -9462.417} C_VEL
LIN {X 0,Y 433.328,Z 568.202,A -85,B 0,C 180,E1 -9463.554,E2 -9463.554} C_VEL
LIN {X 0,Y 433.856,Z 558.137,A -85,B 0,C 180,E1 -9464.422,E2 -9464.422} C_VEL
LIN {X 0,Y 434.712,Z 546.161,A -85,B 0,C 180,E1 -9465.231,E2 -9465.231} C_VEL
LIN {X 0,Y 435.369,Z 533.716,A -85,B 0,C 180,E1 -9465.867,E2 -9465.867} C_VEL
LIN {X 0,Y 435.983,Z 520.976,A -85,B 0,C 180,E1 -9466.325,E2 -9466.325} C_VEL
LIN {X 0,Y 436.293,Z 507.646,A -85,B 0,C 180,E1 -9466.614,E2 -9466.614} C_VEL
LIN {X 0,Y 436.781,Z 437.054,A -85,B 0,C 180,E1 -9467.78,E2 -9467.78} C_VEL
LIN {X 0,Y 433.328,Z 405.21,A -85,B 0,C 180,E1 -9468.472,E2 -9468.472} C_VEL
LIN {X 0,Y 434.025,Z 388.383,A -85,B 0,C 180,E1 -9470.869,E2 -9470.869} C_VEL
LIN {X 0,Y 435.029,Z 367.936,A -85,B 0,C 180,E1 -9473.821,E2 -9473.821} C_VEL
LIN {X 0,Y 436.275,Z 345.655,A -85,B 0,C 180,E1 -9477.053,E2 -9477.053} C_VEL
LIN {X 0,Y 436.709,Z 338.639,A -85,B 0,C 180,E1 -9478.081,E2 -9478.081} C_VEL
LIN {X 0,Y 435.013,Z 329.05,A -85,B 0,C 180,E1 -9479.623,E2 -9479.623} C_VEL
LIN {X 0,Y 432.339,Z 317.729,A -85,B 0,C 180,E1 -9481.583,E2 -9481.583} C_VEL
LIN {X 0,Y 432.323,Z 317.632,A -85,B 0,C 180,E1 -9484.678,E2 -9484.678} C_VEL
LIN {X 0,Y 432.319,Z 317.631,A -85,B 0,C 180,E1 -9488.151,E2 -9488.151} C_VEL
LIN {X 0,Y 432.3,Z 317.638,A -85,B 0,C 180,E1 -9491.8,E2 -9491.8} C_VEL
LIN {X 0,Y 432.328,Z 317.611,A -85,B 0,C 180,E1 -9494.347,E2 -9494.347} C_VEL
LIN {X 0,Y 432.299,Z 317.63,A -85,B 0,C 180,E1 -9497.018,E2 -9497.018} C_VEL
LIN {X 0,Y 432.283,Z 317.634,A -85,B 0,C 180,E1 -9499.827,E2 -9499.827} C_VEL
LIN {X 0,Y 432.29,Z 317.596,A -85,B 0,C 180,E1 -9503.02,E2 -9503.02} C_VEL
LIN {X 0,Y 432.326,Z 317.624,A -85,B 0,C 180,E1 -9506.002,E2 -9506.002} C_VEL
LIN {X 0,Y 432.34,Z 317.63,A -85,B 0,C 180,E1 -9509.49,E2 -9509.49} C_VEL
LIN {X 0,Y 432.336,Z 317.62,A -85,B 0,C 180,E1 -9511.873,E2 -9511.873} C_VEL
LIN {X 0,Y 432.317,Z 317.631,A -85,B 0,C 180,E1 -9514.997,E2 -9514.997} C_VEL
LIN {X 0,Y 432.35,Z 317.615,A -85,B 0,C 180,E1 -9518.045,E2 -9518.045} C_VEL
LIN {X 0,Y 432.377,Z 317.614,A -85,B 0,C 180,E1 -9521.029,E2 -9521.029} C_VEL
LIN {X 0,Y 432.423,Z 317.622,A -85,B 0,C 180,E1 -9523.961,E2 -9523.961} C_VEL
LIN {X 0,Y 432.451,Z 317.611,A -85,B 0,C 180,E1 -9527.803,E2 -9527.803} C_VEL
LIN {X 0,Y 432.454,Z 317.618,A -85,B 0,C 180,E1 -9531.59,E2 -9531.59} C_VEL
LIN {X 0,Y 432.576,Z 317.592,A -85,B 0,C 180,E1 -9534.406,E2 -9534.406} C_VEL
LIN {X 0,Y 432.586,Z 317.597,A -85,B 0,C 180,E1 -9538.138,E2 -9538.138} C_VEL
LIN {X 0,Y 432.611,Z 317.586,A -85,B 0,C 180,E1 -9540,E2 -9540} C_VEL
LIN {X 0,Y 432.561,Z 317.597,A -85,B 0,C 180,E1 -9542.794,E2 -9542.794} C_VEL
LIN {X 0,Y 432.508,Z 317.601,A -85,B 0,C 180,E1 -9546.531,E2 -9546.531} C_VEL
LIN {X 0,Y 432.429,Z 317.613,A -85,B 0,C 180,E1 -9549.353,E2 -9549.353} C_VEL
LIN {X 0,Y 432.424,Z 317.614,A -85,B 0,C 180,E1 -9552.803,E2 -9552.803} C_VEL
LIN {X 0,Y 432.403,Z 317.618,A -85,B 0,C 180,E1 -9556.478,E2 -9556.478} C_VEL
LIN {X 0,Y 432.33,Z 317.624,A -85,B 0,C 180,E1 -9559.961,E2 -9559.961} C_VEL
LIN {X 0,Y 432.304,Z 317.631,A -85,B 0,C 180,E1 -9562.965,E2 -9562.965} C_VEL
LIN {X 0,Y 432.311,Z 317.626,A -85,B 0,C 180,E1 -9566.036,E2 -9566.036} C_VEL
LIN {X 0,Y 432.315,Z 317.605,A -85,B 0,C 180,E1 -9569.19,E2 -9569.19} C_VEL
LIN {X 0,Y 432.316,Z 317.624,A -85,B 0,C 180,E1 -9572.444,E2 -9572.444} C_VEL
LIN {X 0,Y 432.331,Z 317.629,A -85,B 0,C 180,E1 -9575.819,E2 -9575.819} C_VEL
LIN {X 0,Y 432.296,Z 317.615,A -85,B 0,C 180,E1 -9579.349,E2 -9579.349} C_VEL
LIN {X 0,Y 432.299,Z 317.635,A -85,B 0,C 180,E1 -9581.801,E2 -9581.801} C_VEL
LIN {X 0,Y 432.33,Z 317.628,A -85,B 0,C 180,E1 -9584.348,E2 -9584.348} C_VEL
LIN {X 0,Y 432.297,Z 317.62,A -85,B 0,C 180,E1 -9587.019,E2 -9587.019} C_VEL
LIN {X 0,Y 432.285,Z 317.637,A -85,B 0,C 180,E1 -9589.829,E2 -9589.829} C_VEL
LIN {X 0,Y 432.297,Z 317.625,A -85,B 0,C 180,E1 -9593.022,E2 -9593.022} C_VEL
LIN {X 0,Y 432.331,Z 317.628,A -85,B 0,C 180,E1 -9596.003,E2 -9596.003} C_VEL
LIN {X 0,Y 432.337,Z 317.633,A -85,B 0,C 180,E1 -9599.493,E2 -9599.493} C_VEL
LIN {X 0,Y 432.313,Z 317.612,A -85,B 0,C 180,E1 -9601.872,E2 -9601.872} C_VEL
LIN {X 0,Y 432.347,Z 317.633,A -85,B 0,C 180,E1 -9605.548,E2 -9605.548} C_VEL
LIN {X 0,Y 432.349,Z 317.626,A -85,B 0,C 180,E1 -9609.046,E2 -9609.046} C_VEL
LIN {X 0,Y 432.396,Z 317.78,A -85,B 0,C 180,E1 -9611.859,E2 -9611.859} C_VEL
LIN {X 0,Y 432.634,Z 318.817,A -85,B 0,C 180,E1 -9612.023,E2 -9612.023} C_VEL
LIN {X 0,Y 437.589,Z 331.714,A -85,B 0,C 180,E1 -9612.479,E2 -9612.479} C_VEL
LIN {X 0,Y 437.201,Z 398.142,A -85,B 0,C 180,E1 -9613.602,E2 -9613.602} C_VEL
LIN {X 0,Y 437.087,Z 410.855,A -85,B 0,C 180,E1 -9613.987,E2 -9613.987} C_VEL
LIN {X 0,Y 436.807,Z 423.224,A -85,B 0,C 180,E1 -9614.546,E2 -9614.546} C_VEL
LIN {X 0,Y 436.438,Z 435.579,A -85,B 0,C 180,E1 -9615.307,E2 -9615.307} C_VEL
LIN {X 0,Y 435.786,Z 447.164,A -85,B 0,C 180,E1 -9616.239,E2 -9616.239} C_VEL
LIN {X 0,Y 435.197,Z 457.503,A -85,B 0,C 180,E1 -9617.289,E2 -9617.289} C_VEL
LIN {X 0,Y 434.708,Z 465.932,A -85,B 0,C 180,E1 -9618.341,E2 -9618.341} C_VEL
LIN {X 0,Y 434.158,Z 473.691,A -85,B 0,C 180,E1 -9619.507,E2 -9619.507} C_VEL
LIN {X 0,Y 434.044,Z 475.232,A -85,B 0,C 180,E1 -9619.77,E2 -9619.77} C_VEL
LIN {X 0,Y 433.239,Z 477.698,A -85,B 0,C 180,E1 -9620.176,E2 -9620.176} C_VEL
LIN {X 0,Y 430.165,Z 481.547,A -85,B 0,C 180,E1 -9620.788,E2 -9620.788} C_VEL
LIN {X 0,Y 427.102,Z 485.158,A -85,B 0,C 180,E1 -9621.433,E2 -9621.433} C_VEL
LIN {X 0,Y 426.323,Z 487.143,A -85,B 0,C 180,E1 -9621.885,E2 -9621.885} C_VEL
LIN {X 0,Y 426.042,Z 492.381,A -85,B 0,C 180,E1 -9623.369,E2 -9623.369} C_VEL
LIN {X 0,Y 425.612,Z 496.277,A -85,B 0,C 180,E1 -9624.789,E2 -9624.789} C_VEL
LIN {X 0,Y 425.334,Z 499.147,A -85,B 0,C 180,E1 -9626.21,E2 -9626.21} C_VEL
LIN {X 0,Y 425.372,Z 500.5,A -85,B 0,C 180,E1 -9627.159,E2 -9627.159} C_VEL
LIN {X 0,Y 425.225,Z 501.485,A -85,B 0,C 180,E1 -9628.106,E2 -9628.106} C_VEL
LIN {X 0,Y 425.303,Z 502.069,A -85,B 0,C 180,E1 -9629.053,E2 -9629.053} C_VEL
LIN {X 0,Y 425.287,Z 502.299,A -85,B 0,C 180,E1 -9630,E2 -9630} C_VEL
LIN {X 0,Y 425.303,Z 502.115,A -85,B 0,C 180,E1 -9630.947,E2 -9630.947} C_VEL
LIN {X 0,Y 425.225,Z 501.561,A -85,B 0,C 180,E1 -9631.894,E2 -9631.894} C_VEL
LIN {X 0,Y 425.37,Z 500.606,A -85,B 0,C 180,E1 -9632.841,E2 -9632.841} C_VEL
LIN {X 0,Y 425.327,Z 499.302,A -85,B 0,C 180,E1 -9633.79,E2 -9633.79} C_VEL
LIN {X 0,Y 425.606,Z 496.489,A -85,B 0,C 180,E1 -9635.211,E2 -9635.211} C_VEL
LIN {X 0,Y 426.023,Z 492.666,A -85,B 0,C 180,E1 -9636.631,E2 -9636.631} C_VEL
LIN {X 0,Y 426.277,Z 487.591,A -85,B 0,C 180,E1 -9638.103,E2 -9638.103} C_VEL
LIN {X 0,Y 426.898,Z 480.361,A -85,B 0,C 180,E1 -9639.715,E2 -9639.715} C_VEL
LIN {X 0,Y 427.534,Z 472.334,A -85,B 0,C 180,E1 -9641.137,E2 -9641.137} C_VEL
LIN {X 0,Y 428.047,Z 464.116,A -85,B 0,C 180,E1 -9642.324,E2 -9642.324} C_VEL
LIN {X 0,Y 428.594,Z 455.09,A -85,B 0,C 180,E1 -9643.392,E2 -9643.392} C_VEL
LIN {X 0,Y 429.294,Z 444.59,A -85,B 0,C 180,E1 -9644.391,E2 -9644.391} C_VEL
LIN {X 0,Y 429.729,Z 433.096,A -85,B 0,C 180,E1 -9645.267,E2 -9645.267} C_VEL
LIN {X 0,Y 430.146,Z 421.847,A -85,B 0,C 180,E1 -9645.925,E2 -9645.925} C_VEL
LIN {X 0,Y 430.347,Z 408.669,A -85,B 0,C 180,E1 -9646.484,E2 -9646.484} C_VEL
LIN {X 0,Y 430.376,Z 394.927,A -85,B 0,C 180,E1 -9646.849,E2 -9646.849} C_VEL
LIN {X 0,Y 430.874,Z 333.351,A -85,B 0,C 180,E1 -9647.89,E2 -9647.89} C_VEL
LIN {X 0,Y 425.563,Z 319.63,A -85,B 0,C 180,E1 -9648.39,E2 -9648.39} C_VEL
LIN {X 0,Y 425.343,Z 318.599,A -85,B 0,C 180,E1 -9648.577,E2 -9648.577} C_VEL
LIN {X 0,Y 425.292,Z 318.491,A -85,B 0,C 180,E1 -9652.27,E2 -9652.27} C_VEL
LIN {X 0,Y 425.251,Z 318.509,A -85,B 0,C 180,E1 -9655.448,E2 -9655.448} C_VEL
LIN {X 0,Y 425.298,Z 318.492,A -85,B 0,C 180,E1 -9658.857,E2 -9658.857} C_VEL
LIN {X 0,Y 425.245,Z 318.51,A -85,B 0,C 180,E1 -9661.928,E2 -9661.928} C_VEL
LIN {X 0,Y 425.29,Z 318.507,A -85,B 0,C 180,E1 -9665.336,E2 -9665.336} C_VEL
LIN {X 0,Y 425.275,Z 318.509,A -85,B 0,C 180,E1 -9668.9,E2 -9668.9} C_VEL
LIN {X 0,Y 425.251,Z 318.5,A -85,B 0,C 180,E1 -9672.655,E2 -9672.655} C_VEL
LIN {X 0,Y 425.281,Z 318.507,A -85,B 0,C 180,E1 -9675.283,E2 -9675.283} C_VEL
LIN {X 0,Y 425.243,Z 318.509,A -85,B 0,C 180,E1 -9678.617,E2 -9678.617} C_VEL
LIN {X 0,Y 425.273,Z 318.489,A -85,B 0,C 180,E1 -9681.098,E2 -9681.098} C_VEL
LIN {X 0,Y 425.289,Z 318.511,A -85,B 0,C 180,E1 -9684.663,E2 -9684.663} C_VEL
LIN {X 0,Y 425.257,Z 318.504,A -85,B 0,C 180,E1 -9688.072,E2 -9688.072} C_VEL
LIN {X 0,Y 425.289,Z 318.484,A -85,B 0,C 180,E1 -9691.365,E2 -9691.365} C_VEL
LIN {X 0,Y 425.252,Z 318.512,A -85,B 0,C 180,E1 -9694.552,E2 -9694.552} C_VEL
LIN {X 0,Y 425.283,Z 318.504,A -85,B 0,C 180,E1 -9697.73,E2 -9697.73} C_VEL
LIN {X 0,Y 425.353,Z 318.502,A -85,B 0,C 180,E1 -9700.703,E2 -9700.703} C_VEL
LIN {X 0,Y 425.367,Z 318.495,A -85,B 0,C 180,E1 -9703.687,E2 -9703.687} C_VEL
LIN {X 0,Y 425.404,Z 318.49,A -85,B 0,C 180,E1 -9707.598,E2 -9707.598} C_VEL
LIN {X 0,Y 425.388,Z 318.486,A -85,B 0,C 180,E1 -9711.449,E2 -9711.449} C_VEL
LIN {X 0,Y 425.496,Z 318.482,A -85,B 0,C 180,E1 -9714.312,E2 -9714.312} C_VEL
LIN {X 0,Y 425.56,Z 318.471,A -85,B 0,C 180,E1 -9718.107,E2 -9718.107} C_VEL
LIN {X 0,Y 425.5,Z 318.478,A -85,B 0,C 180,E1 -9720.946,E2 -9720.946} C_VEL
LIN {X 0,Y 425.504,Z 318.48,A -85,B 0,C 180,E1 -9722.84,E2 -9722.84} C_VEL
LIN {X 0,Y 425.532,Z 318.469,A -85,B 0,C 180,E1 -9725.687,E2 -9725.687} C_VEL
LIN {X 0,Y 425.397,Z 318.496,A -85,B 0,C 180,E1 -9728.551,E2 -9728.551} C_VEL
LIN {X 0,Y 425.401,Z 318.486,A -85,B 0,C 180,E1 -9732.402,E2 -9732.402} C_VEL
LIN {X 0,Y 425.38,Z 318.5,A -85,B 0,C 180,E1 -9736.312,E2 -9736.312} C_VEL
LIN {X 0,Y 425.321,Z 318.493,A -85,B 0,C 180,E1 -9739.636,E2 -9739.636} C_VEL
LIN {X 0,Y 425.281,Z 318.501,A -85,B 0,C 180,E1 -9742.339,E2 -9742.339} C_VEL
LIN {X 0,Y 425.254,Z 318.511,A -85,B 0,C 180,E1 -9745.448,E2 -9745.448} C_VEL
LIN {X 0,Y 425.306,Z 318.496,A -85,B 0,C 180,E1 -9748.862,E2 -9748.862} C_VEL
LIN {X 0,Y 425.258,Z 318.515,A -85,B 0,C 180,E1 -9751.928,E2 -9751.928} C_VEL
LIN {X 0,Y 425.286,Z 318.5,A -85,B 0,C 180,E1 -9755.337,E2 -9755.337} C_VEL
LIN {X 0,Y 425.271,Z 318.502,A -85,B 0,C 180,E1 -9758.902,E2 -9758.902} C_VEL
LIN {X 0,Y 425.253,Z 318.508,A -85,B 0,C 180,E1 -9762.656,E2 -9762.656} C_VEL
LIN {X 0,Y 425.279,Z 318.485,A -85,B 0,C 180,E1 -9765.284,E2 -9765.284} C_VEL
LIN {X 0,Y 425.244,Z 318.511,A -85,B 0,C 180,E1 -9768.619,E2 -9768.619} C_VEL
LIN {X 0,Y 425.273,Z 318.501,A -85,B 0,C 180,E1 -9771.099,E2 -9771.099} C_VEL
LIN {X 0,Y 425.29,Z 318.501,A -85,B 0,C 180,E1 -9774.664,E2 -9774.664} C_VEL
LIN {X 0,Y 425.32,Z 318.657,A -85,B 0,C 180,E1 -9778.141,E2 -9778.141} C_VEL
LIN {X 0,Y 428.883,Z 334.198,A -85,B 0,C 180,E1 -9780.824,E2 -9780.824} C_VEL
LIN {X 0,Y 429.808,Z 339.52,A -85,B 0,C 180,E1 -9781.694,E2 -9781.694} C_VEL
LIN {X 0,Y 428.6,Z 360.177,A -85,B 0,C 180,E1 -9784.765,E2 -9784.765} C_VEL
LIN {X 0,Y 427.456,Z 380.676,A -85,B 0,C 180,E1 -9787.781,E2 -9787.781} C_VEL
LIN {X 0,Y 426.353,Z 403.906,A -85,B 0,C 180,E1 -9791.189,E2 -9791.189} C_VEL
LIN {X 0,Y 429.995,Z 437.805,A -85,B 0,C 180,E1 -9791.955,E2 -9791.955} C_VEL
LIN {X 0,Y 429.399,Z 510.205,A -85,B 0,C 180,E1 -9793.173,E2 -9793.173} C_VEL
LIN {X 0,Y 429.013,Z 523.807,A -85,B 0,C 180,E1 -9793.525,E2 -9793.525} C_VEL
LIN {X 0,Y 428.317,Z 536.663,A -85,B 0,C 180,E1 -9794.048,E2 -9794.048} C_VEL
LIN {X 0,Y 427.599,Z 548.962,A -85,B 0,C 180,E1 -9794.754,E2 -9794.754} C_VEL
LIN {X 0,Y 426.752,Z 560.078,A -85,B 0,C 180,E1 -9795.577,E2 -9795.577} C_VEL
LIN {X 0,Y 426.089,Z 571.499,A -85,B 0,C 180,E1 -9796.649,E2 -9796.649} C_VEL
LIN {X 0,Y 425.692,Z 579.817,A -85,B 0,C 180,E1 -9797.607,E2 -9797.607} C_VEL
LIN {X 0,Y 425.112,Z 588.457,A -85,B 0,C 180,E1 -9798.799,E2 -9798.799} C_VEL
LIN {X 0,Y 424.736,Z 596.929,A -85,B 0,C 180,E1 -9800.235,E2 -9800.235} C_VEL
LIN {X 0,Y 424.6,Z 603.793,A -85,B 0,C 180,E1 -9801.673,E2 -9801.673} C_VEL
LIN {X 0,Y 424.541,Z 610.096,A -85,B 0,C 180,E1 -9803.346,E2 -9803.346} C_VEL
LIN {X 0,Y 424.626,Z 614.21,A -85,B 0,C 180,E1 -9804.777,E2 -9804.777} C_VEL
LIN {X 0,Y 424.753,Z 617.259,A -85,B 0,C 180,E1 -9806.205,E2 -9806.205} C_VEL
LIN {X 0,Y 424.733,Z 618.701,A -85,B 0,C 180,E1 -9807.155,E2 -9807.155} C_VEL
LIN {X 0,Y 424.976,Z 620.394,A -85,B 0,C 180,E1 -9809.052,E2 -9809.052} C_VEL
LIN {X 0,Y 424.985,Z 620.618,A -85,B 0,C 180,E1 -9810,E2 -9810} C_VEL
LIN {X 0,Y 424.976,Z 620.393,A -85,B 0,C 180,E1 -9810.948,E2 -9810.948} C_VEL
LIN {X 0,Y 424.734,Z 618.701,A -85,B 0,C 180,E1 -9812.845,E2 -9812.845} C_VEL
LIN {X 0,Y 424.753,Z 617.258,A -85,B 0,C 180,E1 -9813.795,E2 -9813.795} C_VEL
LIN {X 0,Y 424.629,Z 614.204,A -85,B 0,C 180,E1 -9815.223,E2 -9815.223} C_VEL
LIN {X 0,Y 424.583,Z 609.935,A -85,B 0,C 180,E1 -9816.702,E2 -9816.702} C_VEL
LIN {X 0,Y 424.6,Z 603.779,A -85,B 0,C 180,E1 -9818.327,E2 -9818.327} C_VEL
LIN {X 0,Y 424.736,Z 596.91,A -85,B 0,C 180,E1 -9819.765,E2 -9819.765} C_VEL
LIN {X 0,Y 425.109,Z 588.433,A -85,B 0,C 180,E1 -9821.201,E2 -9821.201} C_VEL
LIN {X 0,Y 425.681,Z 579.784,A -85,B 0,C 180,E1 -9822.394,E2 -9822.394} C_VEL
LIN {X 0,Y 426.257,Z 569.111,A -85,B 0,C 180,E1 -9823.588,E2 -9823.588} C_VEL
LIN {X 0,Y 426.829,Z 558.582,A -85,B 0,C 180,E1 -9824.542,E2 -9824.542} C_VEL
LIN {X 0,Y 427.72,Z 547.112,A -85,B 0,C 180,E1 -9825.364,E2 -9825.364} C_VEL
LIN {X 0,Y 428.385,Z 535.334,A -85,B 0,C 180,E1 -9826.011,E2 -9826.011} C_VEL
LIN {X 0,Y 429.098,Z 521.817,A -85,B 0,C 180,E1 -9826.533,E2 -9826.533} C_VEL
LIN {X 0,Y 429.477,Z 508.431,A -85,B 0,C 180,E1 -9826.855,E2 -9826.855} C_VEL
LIN {X 0,Y 430.002,Z 437.788,A -85,B 0,C 180,E1 -9828.04,E2 -9828.04} C_VEL
LIN {X 0,Y 426.336,Z 403.941,A -85,B 0,C 180,E1 -9828.803,E2 -9828.803} C_VEL
LIN {X 0,Y 427.433,Z 380.625,A -85,B 0,C 180,E1 -9832.22,E2 -9832.22} C_VEL
LIN {X 0,Y 428.876,Z 355.776,A -85,B 0,C 180,E1 -9835.877,E2 -9835.877} C_VEL
LIN {X 0,Y 429.783,Z 339.464,A -85,B 0,C 180,E1 -9838.308,E2 -9838.308} C_VEL
LIN {X 0,Y 427.693,Z 328.763,A -85,B 0,C 180,E1 -9840.077,E2 -9840.077} C_VEL
LIN {X 0,Y 425.316,Z 318.63,A -85,B 0,C 180,E1 -9841.859,E2 -9841.859} C_VEL
LIN {X 0,Y 425.29,Z 318.501,A -85,B 0,C 180,E1 -9845.336,E2 -9845.336} C_VEL
LIN {X 0,Y 425.273,Z 318.501,A -85,B 0,C 180,E1 -9848.901,E2 -9848.901} C_VEL
LIN {X 0,Y 425.252,Z 318.511,A -85,B 0,C 180,E1 -9852.655,E2 -9852.655} C_VEL
LIN {X 0,Y 425.279,Z 318.485,A -85,B 0,C 180,E1 -9855.283,E2 -9855.283} C_VEL
LIN {X 0,Y 425.244,Z 318.513,A -85,B 0,C 180,E1 -9858.618,E2 -9858.618} C_VEL
LIN {X 0,Y 425.271,Z 318.496,A -85,B 0,C 180,E1 -9861.098,E2 -9861.098} C_VEL
LIN {X 0,Y 425.287,Z 318.49,A -85,B 0,C 180,E1 -9864.663,E2 -9864.663} C_VEL
LIN {X 0,Y 425.258,Z 318.515,A -85,B 0,C 180,E1 -9868.072,E2 -9868.072} C_VEL
LIN {X 0,Y 425.304,Z 318.494,A -85,B 0,C 180,E1 -9871.366,E2 -9871.366} C_VEL
LIN {X 0,Y 425.254,Z 318.511,A -85,B 0,C 180,E1 -9874.552,E2 -9874.552} C_VEL
LIN {X 0,Y 425.285,Z 318.499,A -85,B 0,C 180,E1 -9877.729,E2 -9877.729} C_VEL
LIN {X 0,Y 425.354,Z 318.488,A -85,B 0,C 180,E1 -9880.704,E2 -9880.704} C_VEL
LIN {X 0,Y 425.38,Z 318.5,A -85,B 0,C 180,E1 -9883.688,E2 -9883.688} C_VEL
LIN {X 0,Y 425.404,Z 318.486,A -85,B 0,C 180,E1 -9887.598,E2 -9887.598} C_VEL
LIN {X 0,Y 425.399,Z 318.496,A -85,B 0,C 180,E1 -9891.449,E2 -9891.449} C_VEL
LIN {X 0,Y 425.532,Z 318.47,A -85,B 0,C 180,E1 -9894.313,E2 -9894.313} C_VEL
LIN {X 0,Y 425.555,Z 318.473,A -85,B 0,C 180,E1 -9898.107,E2 -9898.107} C_VEL
LIN {X 0,Y 425.563,Z 318.464,A -85,B 0,C 180,E1 -9900,E2 -9900} C_VEL
LIN {X 0,Y 425.516,Z 318.475,A -85,B 0,C 180,E1 -9902.84,E2 -9902.84} C_VEL
LIN {X 0,Y 425.469,Z 318.477,A -85,B 0,C 180,E1 -9906.64,E2 -9906.64} C_VEL
LIN {X 0,Y 425.389,Z 318.492,A -85,B 0,C 180,E1 -9909.51,E2 -9909.51} C_VEL
LIN {X 0,Y 425.386,Z 318.491,A -85,B 0,C 180,E1 -9912.904,E2 -9912.904} C_VEL
LIN {X 0,Y 425.353,Z 318.496,A -85,B 0,C 180,E1 -9916.604,E2 -9916.604} C_VEL
LIN {X 0,Y 425.321,Z 318.501,A -85,B 0,C 180,E1 -9919.636,E2 -9919.636} C_VEL
LIN {X 0,Y 425.281,Z 318.505,A -85,B 0,C 180,E1 -9922.339,E2 -9922.339} C_VEL
LIN {X 0,Y 425.253,Z 318.513,A -85,B 0,C 180,E1 -9925.448,E2 -9925.448} C_VEL
LIN {X 0,Y 425.293,Z 318.482,A -85,B 0,C 180,E1 -9928.859,E2 -9928.859} C_VEL
LIN {X 0,Y 425.257,Z 318.503,A -85,B 0,C 180,E1 -9931.928,E2 -9931.928} C_VEL
LIN {X 0,Y 425.289,Z 318.512,A -85,B 0,C 180,E1 -9935.337,E2 -9935.337} C_VEL
LIN {X 0,Y 425.273,Z 318.489,A -85,B 0,C 180,E1 -9938.902,E2 -9938.902} C_VEL
LIN {X 0,Y 425.252,Z 318.51,A -85,B 0,C 180,E1 -9942.656,E2 -9942.656} C_VEL
LIN {X 0,Y 425.281,Z 318.503,A -85,B 0,C 180,E1 -9945.284,E2 -9945.284} C_VEL
LIN {X 0,Y 425.244,Z 318.508,A -85,B 0,C 180,E1 -9948.619,E2 -9948.619} C_VEL
LIN {X 0,Y 425.275,Z 318.511,A -85,B 0,C 180,E1 -9951.1,E2 -9951.1} C_VEL
LIN {X 0,Y 425.292,Z 318.506,A -85,B 0,C 180,E1 -9954.664,E2 -9954.664} C_VEL
LIN {X 0,Y 425.252,Z 318.51,A -85,B 0,C 180,E1 -9958.073,E2 -9958.073} C_VEL
LIN {X 0,Y 425.294,Z 318.491,A -85,B 0,C 180,E1 -9961.366,E2 -9961.366} C_VEL
LIN {X 0,Y 425.251,Z 318.511,A -85,B 0,C 180,E1 -9964.552,E2 -9964.552} C_VEL
LIN {X 0,Y 425.292,Z 318.492,A -85,B 0,C 180,E1 -9967.73,E2 -9967.73} C_VEL
LIN {X 0,Y 425.359,Z 318.56,A -85,B 0,C 180,E1 -9971.486,E2 -9971.486} C_VEL
LIN {X 0,Y 425.484,Z 319.311,A -85,B 0,C 180,E1 -9971.679,E2 -9971.679} C_VEL
LIN {X 0,Y 428.793,Z 327.812,A -85,B 0,C 180,E1 -9972.017,E2 -9972.017} C_VEL
LIN {X 0,Y 430.858,Z 333.199,A -85,B 0,C 180,E1 -9972.204,E2 -9972.204} C_VEL
LIN {X 0,Y 430.438,Z 399.144,A -85,B 0,C 180,E1 -9973.337,E2 -9973.337} C_VEL
LIN {X 0,Y 430.323,Z 411.846,A -85,B 0,C 180,E1 -9973.728,E2 -9973.728} C_VEL
LIN {X 0,Y 430.033,Z 424.211,A -85,B 0,C 180,E1 -9974.296,E2 -9974.296} C_VEL
LIN {X 0,Y 429.67,Z 435.463,A -85,B 0,C 180,E1 -9974.992,E2 -9974.992} C_VEL
LIN {X 0,Y 429.036,Z 446.876,A -85,B 0,C 180,E1 -9975.897,E2 -9975.897} C_VEL
LIN {X 0,Y 428.374,Z 457.44,A -85,B 0,C 180,E1 -9976.963,E2 -9976.963} C_VEL
LIN {X 0,Y 427.827,Z 466.913,A -85,B 0,C 180,E1 -9978.151,E2 -9978.151} C_VEL
LIN {X 0,Y 427.25,Z 474.672,A -85,B 0,C 180,E1 -9979.336,E2 -9979.336} C_VEL
LIN {X 0,Y 426.701,Z 482.351,A -85,B 0,C 180,E1 -9980.783,E2 -9980.783} C_VEL
LIN {X 0,Y 426.323,Z 487.143,A -85,B 0,C 180,E1 -9981.885,E2 -9981.885} C_VEL
LIN {X 0,Y 425.521,Z 489.903,A -85,B 0,C 180,E1 -9982.582,E2 -9982.582} C_VEL
LIN {X 0,Y 422.373,Z 494.069,A -85,B 0,C 180,E1 -9983.722,E2 -9983.722} C_VEL
LIN {X 0,Y 419.205,Z 497.615,A -85,B 0,C 180,E1 -9984.911,E2 -9984.911} C_VEL
LIN {X 0,Y 418.384,Z 499.239,A -85,B 0,C 180,E1 -9985.678,E2 -9985.678} C_VEL
LIN {X 0,Y 418.354,Z 501.478,A -85,B 0,C 180,E1 -9987.111,E2 -9987.111} C_VEL
LIN {X 0,Y 418.203,Z 502.463,A -85,B 0,C 180,E1 -9988.074,E2 -9988.074} C_VEL
LIN {X 0,Y 418.28,Z 503.046,A -85,B 0,C 180,E1 -9989.037,E2 -9989.037} C_VEL
LIN {X 0,Y 418.264,Z 503.276,A -85,B 0,C 180,E1 -9990,E2 -9990} C_VEL
LIN {X 0,Y 418.28,Z 503.092,A -85,B 0,C 180,E1 -9990.963,E2 -9990.963} C_VEL
LIN {X 0,Y 418.203,Z 502.538,A -85,B 0,C 180,E1 -9991.926,E2 -9991.926} C_VEL
LIN {X 0,Y 418.351,Z 501.584,A -85,B 0,C 180,E1 -9992.889,E2 -9992.889} C_VEL
LIN {X 0,Y 418.31,Z 500.28,A -85,B 0,C 180,E1 -9993.853,E2 -9993.853} C_VEL
LIN {X 0,Y 418.606,Z 497.466,A -85,B 0,C 180,E1 -9995.298,E2 -9995.298} C_VEL
LIN {X 0,Y 419.043,Z 493.643,A -85,B 0,C 180,E1 -9996.742,E2 -9996.742} C_VEL
LIN {X 0,Y 419.32,Z 488.568,A -85,B 0,C 180,E1 -9998.239,E2 -9998.239} C_VEL
LIN {X 0,Y 419.973,Z 481.336,A -85,B 0,C 180,E1 -9999.876,E2 -9999.876} C_VEL
LIN {X 0,Y 420.641,Z 473.31,A -85,B 0,C 180,E1 -10001.321,E2 -10001.321} C_VEL
LIN {X 0,Y 421.181,Z 465.091,A -85,B 0,C 180,E1 -10002.528,E2 -10002.528} C_VEL
LIN {X 0,Y 421.76,Z 456.064,A -85,B 0,C 180,E1 -10003.613,E2 -10003.613} C_VEL
LIN {X 0,Y 422.49,Z 445.563,A -85,B 0,C 180,E1 -10004.627,E2 -10004.627} C_VEL
LIN {X 0,Y 422.955,Z 434.067,A -85,B 0,C 180,E1 -10005.518,E2 -10005.518} C_VEL
LIN {X 0,Y 423.385,Z 422.818,A -85,B 0,C 180,E1 -10006.186,E2 -10006.186} C_VEL
LIN {X 0,Y 423.599,Z 409.635,A -85,B 0,C 180,E1 -10006.754,E2 -10006.754} C_VEL
LIN {X 0,Y 423.632,Z 395.886,A -85,B 0,C 180,E1 -10007.125,E2 -10007.125} C_VEL
